// TwinCAT 3 PLC project TwinCAT_OpenFramework_Temporary
// Title: Temporary project for old code storing
// Company: Oleksandr Tiutyk FOP
// ProjectVersion: 0.0.0.1
// Description: Temporary project that contains legacy functionality and needs to be reconsidered and migrated in light of the new concepts
// ProgramVersion: 3.1.4026.16
// project tree:
//   Communication/ADS/ AdsCommunicationSettings.TcPOU, AdsCommunicator.TcPOU, ADS_COMMUNICATOR_STATE.TcDUT, ADS_REQUEST_ITEM.TcDUT
//   Communication/ CommunicationSettings.TcPOU, Communicator.TcPOU, CommunicatorSFC.TcPOU, CurrentNamespace_1.TcGVL
//   Communication/OPC_UA/ OpcUaCommunicationSettings.TcPOU, OpcUaCommunicator.TcPOU, OpcUaHelper.TcPOU, OPC_UA_ACTION_EXECUTION_STATE.TcDUT, OPC_UA_COMMUNICATOR_STATE.TcDUT
//   Communication/OPC_UA/RequestItems/ OpcUaDAReadRequestItem.TcPOU, OpcUaDARequestItem.TcPOU, OpcUaDAWriteRequestItem.TcPOU, OpcUaMethodCallRequestItem.TcPOU, OpcUaRequestItem.TcPOU, OPC_UA_OUTPUT_ARGUMENT_INFO_AND_DATA.TcDUT
//   Communication/S7/ GetStringSizeForS7Comm.TcPOU, S7CommunicationSettings.TcPOU, S7Communicator.TcPOU, S7_COMMUNICATOR_STATE.TcDUT, S7_VARIABLE.TcDUT
//   Database/Command/ DbCommandExecutor.TcPOU, DB_COMMAND_DISCONNECTING_STATE.TcDUT, DB_COMMAND_EXECUTION_PARAMETERS.TcDUT, DB_COMMAND_EXECUTION_STATE.TcDUT
//   Database/ CurrentNamespace.TcGVL
//   Database/StoredProcedure/ DbProcedureExecutor.TcPOU, DB_PROCEDURE_DISCONNECTING_STATE.TcDUT, DB_PROCEDURE_EXECUTION_STATE.TcDUT, DB_ROCEDURE_EXECUTION_PARAMETERS.TcDUT
//   Files/ CreateDirectory.TcPOU, DeleteDirectory.TcPOU, DeleteFile.TcPOU, LoadFile.TcPOU, RenameFile.TcPOU
//   Files/FileContentManager/Enums/ FILE_CONTENT_HANDLING_MODE.TcDUT, FILE_MOVE_POINTER_TYPE.TcDUT, FILE_OPEN_MODE.TcDUT
//   Files/FileContentManager/ FileContentManager.TcPOU, FileContentTask.TcPOU
//   Files/FileContentManager/Tasks/ FileCloseTask.TcPOU, FileFlushTask.TcPOU, FileGetCurrentPositionTask.TcPOU, FileMovePointerTask.TcPOU, FileOpenTask.TcPOU, FileReadBytesTask.TcPOU, FileReadStringTask.TcPOU, FileTestForEndTask.TcPOU, FileWriteBytesTask.TcPOU, FileWriteStringTask.TcPOU
//   StateMachine/Finite/ FiniteStateMachine.TcPOU, ProgramState.TcPOU, ProgramTransition.TcPOU
//   StateMachine/ ProgramConstants.TcGVL
//   StateMachine/Program/ ProgramStateMachine.TcPOU
//   StateMachine/Program/States/ HaltedProgramState.TcPOU, ReadyProgramState.TcPOU, RunningProgramState.TcPOU, SuspendedProgramState.TcPOU
//   StateMachine/Program/Transitions/ HaltedToReadyProgramTransition.TcPOU, ReadyToHaltedProgramTransition.TcPOU, ReadyToRunningProgramTransition.TcPOU, RunningToHaltedProgramTransition.TcPOU, RunningToReadyProgramTransition.TcPOU, RunningToSuspendedProgramTransition.TcPOU, SuspendedToHaltedProgramTransition.TcPOU, SuspendedToReadyProgramTransition.TcPOU, SuspendedToRunningProgramTransition.TcPOU
//   StateMachine/UnifiedProgram/States/ HaltedUnifiedProgramState.TcPOU, ReadyUnifiedProgramState.TcPOU, RunningUnifiedProgramState.TcPOU, SuspendedUnifiedProgramState.TcPOU
//   StateMachine/UnifiedProgram/StepModels/ UnifiedProgramExecutedStep.TcPOU, UnifiedProgramExecutedStepAction.TcPOU, UnifiedProgramExecutedStepHelper.TcPOU, UnifiedProgramExecutedStepTransition.TcPOU, UnifiedProgramExecutedStepTransitionCondition.TcPOU
//   StateMachine/UnifiedProgram/Steps/ UNIFIED_PROGRAM_CONFIGURATION.TcDUT, UNIFIED_PROGRAM_EXECUTED_STEP.TcDUT, UNIFIED_PROGRAM_STEP.TcDUT, UNIFIED_PROGRAM_STEP_ACTION.TcDUT, UNIFIED_PROGRAM_STEP_TRANSITION.TcDUT, UNIFIED_PROGRAM_STEP_TRANSITION_CONDITION.TcDUT
//   StateMachine/UnifiedProgram/Transitions/ HaltedToReadyUnifiedProgramTransition.TcPOU, ReadyToHaltedUnifiedProgramTransition.TcPOU, ReadyToRunningUnifiedProgramTransition.TcPOU, RunningToHaltedUnifiedProgramTransition.TcPOU, RunningToReadyUnifiedProgramTransition.TcPOU, RunningToSuspendedUnifiedProgramTransition.TcPOU, SuspendedToHaltedUnifiedProgramTransition.TcPOU, SuspendedToReadyUnifiedProgramTransition.TcPOU, SuspendedToRunningUnifiedProgramTransition.TcPOU
//   StateMachine/UnifiedProgram/ UnifiedProgramConstants.TcGVL, UnifiedProgramStateMachine.TcPOU, UnifiedProgramStepExecutor.TcPOU
//   Tasks/ SequentialTaskExecutor.TcPOU, Task.TcPOU

// ---- Communication/ADS/ADS_COMMUNICATOR_STATE.TcDUT
{attribute 'qualified_only'}
{attribute 'strict'}
{attribute 'to_string'}
TYPE ADS_COMMUNICATOR_STATE :
(
	IDLE_OR_DONE,
	READ_SYMBOL_INFO,
	DATA_PROCESSING,
	WAIT_FOR_NEXT_CYCLE
);
END_TYPE

// ---- Communication/ADS/ADS_REQUEST_ITEM.TcDUT
{attribute 'enable_dynamic_creation'}	
TYPE ADS_REQUEST_ITEM :
STRUCT
	ReadSymbolInfo : Tc2_Utilities.PLC_ReadSymInfoByName;
	ReadMode : BOOL;
	Read : Tc2_System.ADSREADEX;
	Write : Tc2_System.ADSWRITE;
	IndexGroupAndOffsetValid : BOOL;	
	ReceivedBytesCountTarget : POINTER TO UDINT;
END_STRUCT
END_TYPE

// ---- Communication/OPC_UA/OPC_UA_ACTION_EXECUTION_STATE.TcDUT
{attribute 'qualified_only'}
{attribute 'strict'}
{attribute 'to_string'}
TYPE OPC_UA_ACTION_EXECUTION_STATE :
(
	BUSY,
	DONE,
	ERROR
);
END_TYPE

// ---- Communication/OPC_UA/OPC_UA_COMMUNICATOR_STATE.TcDUT
{attribute 'qualified_only'}
{attribute 'strict'}
{attribute 'to_string'}
TYPE OPC_UA_COMMUNICATOR_STATE :
(
	IDLE,
	CONNECT,
	GET_NAMESPACE_INDEX,
	GET_NODE_HANDLE,
	PERFORM_ACTION,
	WAIT_FOR_NEXT_CYCLE,
	RELEASE_NODE_HANDLE,
	DISCONNECT
);
END_TYPE

// ---- Communication/OPC_UA/RequestItems/OPC_UA_OUTPUT_ARGUMENT_INFO_AND_DATA.TcDUT
{attribute 'pack_mode' := '1'}
TYPE OPC_UA_OUTPUT_ARGUMENT_INFO_AND_DATA :
STRUCT
	nNumberOfOutputArguments: UDINT; // determined amount of output parameters
	nReserved: ARRAY[1..4] OF BYTE; // Reserved padding
	//stOutputArgInfo: ARRAY[*] OF ST_UAMethodArgInfo; 
	//data : DINT;
END_STRUCT
END_TYPE

// ---- Communication/S7/S7_COMMUNICATOR_STATE.TcDUT
{attribute 'qualified_only'}
{attribute 'strict'}
{attribute 'to_string'}
TYPE S7_COMMUNICATOR_STATE :
(
	IDLE_OR_DONE,
	DATA_PROCESSING,
	WAIT_FOR_NEXT_CYCLE
);
END_TYPE

// ---- Communication/S7/S7_VARIABLE.TcDUT
{attribute 'enable_dynamic_creation'}	
TYPE S7_VARIABLE :
STRUCT
	Address : PVOID;
	Write : BOOL;
END_STRUCT
END_TYPE

// ---- Database/Command/DB_COMMAND_DISCONNECTING_STATE.TcDUT
{attribute 'qualified_only'}
{attribute 'strict'}
{attribute 'to_string'}
TYPE DB_COMMAND_DISCONNECTING_STATE :
(
	IDLING,
	DATA_SET_RELEASING,
	DISCONNECTING
);
END_TYPE

// ---- Database/Command/DB_COMMAND_EXECUTION_PARAMETERS.TcDUT
{attribute 'enable_dynamic_creation'}	
TYPE DB_COMMAND_EXECUTION_PARAMETERS :
STRUCT
	DbId : UDINT;
	CommandText : Tc2_System.T_MaxString;
	TargetBuffer : PVOID; 
	TargetBufferSize : UDINT;
	MaxRecordsToReadAtTime : UINT;
END_STRUCT
END_TYPE

// ---- Database/Command/DB_COMMAND_EXECUTION_STATE.TcDUT
{attribute 'qualified_only'}
{attribute 'strict'}
{attribute 'to_string'}
TYPE DB_COMMAND_EXECUTION_STATE :
(
	IDLING,
	STARTING,
	CONNECTING,
	PREPARING,
	EXECUTING,
	LOADING_RESULT_DATA_SET,
	DISCONNECTING 
);
END_TYPE

// ---- Database/StoredProcedure/DB_PROCEDURE_DISCONNECTING_STATE.TcDUT
{attribute 'qualified_only'}
{attribute 'strict'}
{attribute 'to_string'}
TYPE DB_PROCEDURE_DISCONNECTING_STATE :
(
	IDLING,
	DATA_SET_RELEASING,
	PARAMETERS_RELEASING,
	DISCONNECTING
);
END_TYPE

// ---- Database/StoredProcedure/DB_PROCEDURE_EXECUTION_STATE.TcDUT
{attribute 'qualified_only'}
{attribute 'strict'}
{attribute 'to_string'}
TYPE DB_PROCEDURE_EXECUTION_STATE :
(
	IDLING,
	STARTING,
	CONNECTING,
	PREPARING,
	EXECUTING,
	LOADING_RESULT_DATA_SET,
	DISCONNECTING
);
END_TYPE

// ---- Database/StoredProcedure/DB_ROCEDURE_EXECUTION_PARAMETERS.TcDUT
{attribute 'enable_dynamic_creation'}	
TYPE DB_ROCEDURE_EXECUTION_PARAMETERS :
STRUCT
	DbId : UDINT;
	ProcedureName : Tc2_System.T_MaxString;
	ParameterDescriptors : POINTER TO Tc3_Database.ST_SQLSPParameter;
	ParameterDescriptorsSize : UDINT;
	ParameterValues : PVOID;
	ParameterValuesSize : UDINT;	
	TargetBuffer : PVOID; 
	TargetBufferSize : UDINT;
	MaxRecordsToReadAtTime : UINT;
END_STRUCT
END_TYPE

// ---- Files/FileContentManager/Enums/FILE_CONTENT_HANDLING_MODE.TcDUT
{attribute 'qualified_only'}
{attribute 'strict'}
{attribute 'to_string'}
TYPE FILE_CONTENT_HANDLING_MODE :
(
	BINARY := Tc2_System.FOPEN_MODEBINARY, // opens the file in binary mode
	TEXT := Tc2_System.FOPEN_MODETEXT // opens the file in text mode
) DWORD;
END_TYPE

// ---- Files/FileContentManager/Enums/FILE_MOVE_POINTER_TYPE.TcDUT
{attribute 'qualified_only'}
{attribute 'strict'}
{attribute 'to_string'}
TYPE FILE_MOVE_POINTER_TYPE :
(
	FROM_FILE_BEGINNING,
	FROM_CURRENT_POSITION,
	FROM_FILE_END
);
END_TYPE

// ---- Files/FileContentManager/Enums/FILE_OPEN_MODE.TcDUT
{attribute 'qualified_only'}
{attribute 'strict'}
{attribute 'to_string'}
TYPE FILE_OPEN_MODE :
(
	READ_EXISTING := Tc2_System.FOPEN_MODEREAD, // opens a file for reading. An error is returned if the file cannot be found or does not exist
	WRITE_EMPTY := Tc2_System.FOPEN_MODEWRITE, // opens an empty file for writing. If the file already exists, it is overwritten
	APPEND := Tc2_System.FOPEN_MODEAPPEND, // opens a file for writing at the end of the file (append). If the file does not exist, a new file is created
	READ_AND_WRITE_EXISTING := Tc2_System.FOPEN_MODEREAD OR Tc2_System.FOPEN_MODEPLUS, // opens a file for reading and writing. The file must exist
	READ_AND_WRITE_EMPTY := Tc2_System.FOPEN_MODEWRITE OR Tc2_System.FOPEN_MODEPLUS, // opens an empty file FOR reading AND writing. IF the file already exists, it is overwritten.
	READ_AND_APPEND := Tc2_System.FOPEN_MODEAPPEND OR Tc2_System.FOPEN_MODEPLUS // opens a file for reading and writing at the end of the file (append). If the file does not exist, a new file is created. For this, the memory path must be known, otherwise error 1804 appears.
) DWORD;
END_TYPE

// ---- StateMachine/UnifiedProgram/Steps/UNIFIED_PROGRAM_CONFIGURATION.TcDUT
TYPE UNIFIED_PROGRAM_CONFIGURATION :
STRUCT
	Name : STRING(255) := 'New program';
	Version : DATE_AND_TIME;
	Steps : ARRAY [0..UnifiedProgramConstants.MaxStepCount - 1] OF UNIFIED_PROGRAM_STEP;
END_STRUCT
END_TYPE

// ---- StateMachine/UnifiedProgram/Steps/UNIFIED_PROGRAM_EXECUTED_STEP.TcDUT
TYPE UNIFIED_PROGRAM_EXECUTED_STEP :
STRUCT
	StepIndex : INT := -1;
	
	Step : REFERENCE TO UNIFIED_PROGRAM_STEP;
END_STRUCT
END_TYPE

// ---- StateMachine/UnifiedProgram/Steps/UNIFIED_PROGRAM_STEP.TcDUT
TYPE UNIFIED_PROGRAM_STEP :
STRUCT
	Suspend : BOOL;
	Complete : BOOL;
	Actions : ARRAY [0..UnifiedProgramConstants.MaxStepActionsCount - 1] OF UNIFIED_PROGRAM_STEP_ACTION;
	Transitions : ARRAY [0..UnifiedProgramConstants.MaxStepTransitionsCount - 1] OF UNIFIED_PROGRAM_STEP_TRANSITION;
END_STRUCT
END_TYPE

// ---- StateMachine/UnifiedProgram/Steps/UNIFIED_PROGRAM_STEP_ACTION.TcDUT
TYPE UNIFIED_PROGRAM_STEP_ACTION :
STRUCT
	Name : STRING;
	Args : ARRAY [0..UnifiedProgramConstants.MaxActionArgumentsCount - 1] OF STRING(255);
END_STRUCT
END_TYPE

// ---- StateMachine/UnifiedProgram/Steps/UNIFIED_PROGRAM_STEP_TRANSITION.TcDUT
TYPE UNIFIED_PROGRAM_STEP_TRANSITION :
STRUCT
	Condition : UNIFIED_PROGRAM_STEP_TRANSITION_CONDITION;
	Target : BYTE;
END_STRUCT
END_TYPE

// ---- StateMachine/UnifiedProgram/Steps/UNIFIED_PROGRAM_STEP_TRANSITION_CONDITION.TcDUT
TYPE UNIFIED_PROGRAM_STEP_TRANSITION_CONDITION :
STRUCT
	Name : STRING;
	Args : ARRAY [0..UnifiedProgramConstants.MaxActionArgumentsCount - 1] OF STRING(255);
END_STRUCT
END_TYPE

// ---- Communication/CurrentNamespace_1.TcGVL
{attribute 'qualified_only'}
VAR_GLOBAL
	{attribute 'OPC.UA.DA' := '1'}
	{attribute 'OPC.UA.DA.Access' := '1'}
	{attribute 'init_namespace'} 
	Name : STRING(255);	
END_VAR

// ---- Database/CurrentNamespace.TcGVL
{attribute 'qualified_only'}
VAR_GLOBAL
	{attribute 'OPC.UA.DA' := '1'}
	{attribute 'OPC.UA.DA.Access' := '1'}
	{attribute 'init_namespace'} 
	Name : STRING(255);	
END_VAR

// ---- StateMachine/ProgramConstants.TcGVL
{attribute 'qualified_only'}
VAR_GLOBAL CONSTANT
	MaxStateCount : INT := 5;
	MaxTransitionCount : INT := 20;
END_VAR

// ---- StateMachine/UnifiedProgram/UnifiedProgramConstants.TcGVL
{attribute 'qualified_only'}
VAR_GLOBAL CONSTANT
	MaxStepCount : INT := 5;	
	MaxStepActionsCount : INT := 5;
	MaxStepTransitionsCount : INT := 2;
	MaxActionArgumentsCount : INT := 5;
	MaxConditionArgumentsCount : INT := 5;
END_VAR

// ---- Communication/ADS/AdsCommunicationSettings.TcPOU
{attribute 'no_explicit_call' := 'do not call this function block directly'} 
FUNCTION_BLOCK AdsCommunicationSettings EXTENDS CommunicationSettings
VAR_INPUT
	AmsNetId : Tc2_System.T_AmsNetID;
	AmsPort : Tc2_System.T_AmsPort := 801;
END_VAR
VAR
	_ClassName : STRING := __POUNAME();
END_VAR

PROPERTY CommunicationTypeName : STRING
GET
CommunicationTypeName := 'ADS';
END_GET
END_PROPERTY

END_FUNCTION_BLOCK

// ---- Communication/CommunicationSettings.TcPOU
FUNCTION_BLOCK ABSTRACT CommunicationSettings
VAR_INPUT
	DefaultOperationTimeout : TIME := Tc2_System.DEFAULT_ADS_TIMEOUT;
END_VAR

PROPERTY ABSTRACT CommunicationTypeName : STRING
GET
END_GET
END_PROPERTY

END_FUNCTION_BLOCK

// ---- Communication/ADS/AdsCommunicator.TcPOU
{attribute 'no_explicit_call' := 'do not call this function block directly'} 
FUNCTION_BLOCK AdsCommunicator EXTENDS Communicator
VAR
	{attribute 'OPC.UA.DA' := '0'}	
	_ClassName : STRING := __POUNAME();

	{attribute 'OPC.UA.DA' := '0'}	
	_State : ADS_COMMUNICATOR_STATE;
	{attribute 'OPC.UA.DA' := '0'}	
	_DataProcessed : BOOL;

	{attribute 'OPC.UA.DA' := '0'}
	_Items : List(POINTER_TYPE.STRUCT_POINTER); // of ADS_REQUEST_ITEM 

	{attribute 'OPC.UA.DA' := '0'}	
	_OperationTimer : Timer;	
END_VAR

METHOD AddReadByIndexGroupAndOffset : DINT
VAR_INPUT
	indexGroup : UDINT;
	indexOffset : UDINT;
	targetVariable : __SYSTEM.AnyType;
	receivedBytesCountTarget : POINTER TO UDINT;
	operationTimeout : TIME := T#0S;
END_VAR
VAR_OUTPUT
	exception : Exception;
END_VAR
VAR
	request : POINTER TO ADS_REQUEST_ITEM;
END_VAR
AddReadByIndexGroupAndOffset := -1;

IF Busy THEN
	ExceptionHelper.Throw(0, "AdsRequest is already executing", __POUNAME(), ClassName, CurrentNamespace.Name, __POSITION());
	RETURN;
END_IF

request := __NEW(ADS_REQUEST_ITEM);

request^.ReadMode := TRUE;
request^.ReadSymbolInfo.SYMNAME := '';
request^.Read.IDXGRP := indexGroup;
request^.Read.IDXOFFS := indexOffset;
request^.Read.DESTADDR := targetVariable.pValue;
request^.Read.LEN := TO_UDINT(targetVariable.diSize);
request^.Read.TMOUT := GetOperationTimeout(operationTimeout);
request^.IndexGroupAndOffsetValid := TRUE;
request^.ReceivedBytesCountTarget := receivedBytesCountTarget;

AddReadByIndexGroupAndOffset := _Items.Append(request);
END_METHOD

METHOD AddReadBySymbolName : DINT
VAR_INPUT
	symbolName : Tc2_System.T_MaxString;
	targetVariable : __SYSTEM.AnyType;
	receivedBytesCountTarget : POINTER TO UDINT;
	operationTimeout : TIME := T#0S;
END_VAR
VAR_OUTPUT
	exception : Exception;
END_VAR
VAR
	request : POINTER TO ADS_REQUEST_ITEM;
END_VAR
AddReadBySymbolName := -1;

IF Busy THEN
	ExceptionHelper.Throw(0, "AdsRequest is already executing", __POUNAME(), ClassName, CurrentNamespace.Name, __POSITION());
	RETURN;
END_IF

IF SymbolName = '' THEN
	ExceptionHelper.Throw(0, "Parameter 'symbolName' is not specified", __POUNAME(), ClassName, CurrentNamespace.Name, __POSITION());
	RETURN;
END_IF

request := __NEW(ADS_REQUEST_ITEM);

request^.ReadMode := TRUE;
request^.ReadSymbolInfo.SYMNAME := symbolName;
request^.Read.IDXGRP := 0;
request^.Read.IDXOFFS := 0;
request^.Read.DESTADDR := targetVariable.pValue;
request^.Read.LEN := TO_UDINT(targetVariable.diSize);
request^.Read.TMOUT := GetOperationTimeout(operationTimeout);
request^.IndexGroupAndOffsetValid := FALSE;
request^.ReceivedBytesCountTarget := receivedBytesCountTarget;

AddReadBySymbolName := _Items.Append(request);
END_METHOD

METHOD AddWriteByIndexGroupAndOffset : DINT
VAR_INPUT
	indexGroup : UDINT;
	indexOffset : UDINT;
	sourceVariable : __SYSTEM.AnyType;
	operationTimeout : TIME := T#0S;
END_VAR
VAR_OUTPUT
	exception : Exception;
END_VAR
VAR
	request : POINTER TO ADS_REQUEST_ITEM;
END_VAR
AddWriteByIndexGroupAndOffset := -1;

IF Busy THEN
	ExceptionHelper.Throw(0, "AdsRequest is already executing", __POUNAME(), ClassName, CurrentNamespace.Name, __POSITION());
	RETURN;
END_IF

request := __NEW(ADS_REQUEST_ITEM);

request^.ReadMode := FALSE;
request^.ReadSymbolInfo.SYMNAME := '';
request^.Write.IDXGRP := indexGroup;
request^.Write.IDXOFFS := indexOffset;
request^.Write.SRCADDR := sourceVariable.pValue;
request^.Write.LEN := TO_UDINT(sourceVariable.diSize);
request^.Write.TMOUT := GetOperationTimeout(operationTimeout);
request^.IndexGroupAndOffsetValid := TRUE;

AddWriteByIndexGroupAndOffset := _Items.Append(request);
END_METHOD

METHOD AddWriteBySymbolName : DINT
VAR_INPUT
	symbolName : Tc2_System.T_MaxString;
	sourceVariable : __SYSTEM.AnyType;
	operationTimeout : TIME := T#0S;
END_VAR
VAR_OUTPUT
	exception : Exception;
END_VAR
VAR
	request : POINTER TO ADS_REQUEST_ITEM;
END_VAR
AddWriteBySymbolName := -1;

IF Busy THEN
	ExceptionHelper.Throw(0, "AdsRequest is already executing", __POUNAME(), ClassName, CurrentNamespace.Name, __POSITION());
	RETURN;
END_IF

IF SymbolName = '' THEN
	ExceptionHelper.Throw(0, "Parameter 'symbolName' is not specified", __POUNAME(), ClassName, CurrentNamespace.Name, __POSITION());
	RETURN;
END_IF

request := __NEW(ADS_REQUEST_ITEM);

request^.ReadMode := FALSE;
request^.ReadSymbolInfo.SYMNAME := symbolName;
request^.Write.IDXGRP := 0;
request^.Write.IDXOFFS := 0;
request^.Write.SRCADDR := sourceVariable.pValue;
request^.Write.LEN := TO_UDINT(sourceVariable.diSize);
request^.Write.TMOUT := GetOperationTimeout(operationTimeout);
request^.IndexGroupAndOffsetValid := FALSE;

AddWriteBySymbolName := _Items.Append(request);
END_METHOD

{attribute 'monitoring' := 'call'}
{attribute 'OPC.UA.DA' := '1'}
{attribute 'OPC.UA.DA.Property' := '1'}
PROPERTY Busy : BOOL
GET
Busy := _LastException.Empty AND_THEN _State <> ADS_COMMUNICATOR_STATE.IDLE_OR_DONE;
END_GET
END_PROPERTY

{attribute 'monitoring' := 'call'}
PROPERTY ClassName : STRING
GET
ClassName := _ClassName;
END_GET
END_PROPERTY

PROPERTY CommunicationTypeName : STRING
GET
CommunicationTypeName := 'ADS';
END_GET
END_PROPERTY

{attribute 'monitoring' := 'call'}
{attribute 'OPC.UA.DA' := '1'}
{attribute 'OPC.UA.DA.Property' := '1'}
PROPERTY DataProcessed : BOOL
GET
DataProcessed := _DataProcessed;
END_GET
END_PROPERTY

{attribute 'monitoring' := 'call'}
{attribute 'OPC.UA.DA' := '1'}
{attribute 'OPC.UA.DA.Property' := '1'}
PROPERTY Error : BOOL
GET
Error := NOT _LastException.Empty;
END_GET
END_PROPERTY

METHOD Execute 
VAR
	i : DINT;
	readyItemsCount : DINT;
	item : POINTER TO ADS_REQUEST_ITEM;
END_VAR
_DataProcessed := FALSE;
_OperationTimer.Execute();

StateMachine:

readyItemsCount := 0;

CASE _State OF
	ADS_COMMUNICATOR_STATE.READ_SYMBOL_INFO:
		FOR i := 0 TO _Items.Count - 1 DO
			item := _Items.Get(i); 
			
			IF NOT item^.IndexGroupAndOffsetValid THEN
				item^.ReadSymbolInfo(START := TRUE);
				
				IF item^.ReadSymbolInfo.ERR THEN
					_LastExceptionHelper.Throw(item^.ReadSymbolInfo.ERRID, WStringHelper.Concat2("Execution of PLC_ReadSymInfoByName failed with error id = ", TO_WSTRING(item^.ReadSymbolInfo.ERRID)), __POUNAME(), ClassName, CurrentNamespace.Name, __POSITION());	
					_State := ADS_COMMUNICATOR_STATE.IDLE_OR_DONE;
					RETURN;
				ELSIF NOT item^.ReadSymbolInfo.BUSY THEN
					IF item^.ReadMode THEN
						item^.Read.IDXGRP := item^.ReadSymbolInfo.SYMINFO.idxGroup;
						item^.Read.IDXOFFS := item^.ReadSymbolInfo.SYMINFO.idxOffset;
					ELSE
						item^.Write.IDXGRP := item^.ReadSymbolInfo.SYMINFO.idxGroup;
						item^.Write.IDXOFFS := item^.ReadSymbolInfo.SYMINFO.idxOffset;
					END_IF		

					item^.IndexGroupAndOffsetValid := TRUE;	
					readyItemsCount := readyItemsCount + 1;
				END_IF
			ELSE
				readyItemsCount := readyItemsCount + 1;
			END_IF
		END_FOR
		
		IF readyItemsCount = _Items.Count THEN	
			_State := ADS_COMMUNICATOR_STATE.DATA_PROCESSING;				
			_OperationTimer.Start();
			JMP StateMachine;
		END_IF		
		
	ADS_COMMUNICATOR_STATE.DATA_PROCESSING:
		FOR i := 0 TO _Items.Count - 1 DO
			item := _Items.Get(i); 
			
			IF item^.ReadMode THEN
				item^.Read(READ := TRUE);
				
				IF item^.Read.ERR THEN
					_LastExceptionHelper.Throw(item^.Read.ERRID, WStringHelper.Concat2("Execution of ADSREADEX failed with error id = ", TO_WSTRING(item^.Read.ERRID)), __POUNAME(), ClassName, CurrentNamespace.Name, __POSITION());
					_State := ADS_COMMUNICATOR_STATE.IDLE_OR_DONE;
					RETURN;
				ELSIF NOT item^.Read.BUSY THEN
					IF item^.ReceivedBytesCountTarget <> 0 THEN
						item^.ReceivedBytesCountTarget^ := item^.Read.COUNT_R;
					END_IF
					
					readyItemsCount := readyItemsCount + 1;
				END_IF
			ELSE
				item^.Write(WRITE := TRUE);
				
				IF item^.Write.ERR THEN
					_LastExceptionHelper.Throw(item^.Write.ERRID, WStringHelper.Concat2("Execution of ADSWRITE failed with error id = ", TO_WSTRING(item^.Write.ERRID)), __POUNAME(), ClassName, CurrentNamespace.Name, __POSITION());
					_State := ADS_COMMUNICATOR_STATE.IDLE_OR_DONE;
					RETURN;
				ELSIF NOT item^.Write.BUSY THEN
					readyItemsCount := readyItemsCount + 1;
				END_IF
			END_IF
		END_FOR
		
		IF readyItemsCount = _Items.Count THEN
			_DataProcessed := TRUE;	
			CycleCount := CycleCount + 1;
			
			IF CyclicMode THEN
				_State := ADS_COMMUNICATOR_STATE.WAIT_FOR_NEXT_CYCLE;	
				JMP StateMachine;			
			ELSE	
				_State := ADS_COMMUNICATOR_STATE.IDLE_OR_DONE;		
			END_IF
		END_IF	
		
	ADS_COMMUNICATOR_STATE.WAIT_FOR_NEXT_CYCLE:
		IF _OperationTimer.ElapsedTime >= CycleInterval THEN
			FOR i := 0 TO _Items.Count - 1 DO
				item := _Items.Get(i); 
				
				IF item^.ReadMode THEN
					item^.Read(READ := FALSE);
				ELSE
					item^.Write(WRITE := FALSE);
				END_IF
			END_FOR	
			
			_State := ADS_COMMUNICATOR_STATE.DATA_PROCESSING;
			_OperationTimer.Start();			
			JMP StateMachine;	
		END_IF
END_CASE
END_METHOD

METHOD FB_exit : BOOL
VAR_INPUT
	bInCopyCode : BOOL; // if TRUE, the exit method is called for exiting an instance that is copied afterwards (online change).
END_VAR
_Items.Clear(TRUE);
END_METHOD

METHOD PROTECTED InternalClear : BOOL
VAR_OUTPUT
	exception : Exception;
END_VAR
_Items.Clear(TRUE);

_State := ADS_COMMUNICATOR_STATE.IDLE_OR_DONE;

InternalClear := TRUE;
END_METHOD

METHOD PROTECTED InternalConfigure : BOOL
VAR_INPUT
	settings : REFERENCE TO CommunicationSettings;
END_VAR
VAR_OUTPUT
	exception : Exception;
END_VAR
VAR
	adsSettings : POINTER TO AdsCommunicationSettings;
	i : DINT;
	item : POINTER TO ADS_REQUEST_ITEM;
END_VAR
adsSettings := ADR(settings);

_OperationTimer.Interval := T#1H;

IF adsSettings^.AmsPort = 0 THEN
	ExceptionHelper.Throw(0, "settings.AmsPort is not specified", __POUNAME(), ClassName, CurrentNamespace.Name, __POSITION());
	RETURN;
END_IF

FOR i := 0 TO _Items.Count - 1 DO
	item := _Items.Get(i);
	
	item^.ReadSymbolInfo(NETID := adsSettings^.AmsNetId, PORT := adsSettings^.AmsPort);		
	item^.Read(NETID := adsSettings^.AmsNetId, PORT := adsSettings^.AmsPort);
	item^.Write(NETID := adsSettings^.AmsNetId, PORT := adsSettings^.AmsPort);
END_FOR

InternalConfigure := TRUE;
END_METHOD

METHOD PROTECTED InternalStart : BOOL
VAR_OUTPUT
	exception : Exception;
END_VAR
VAR
	i : DINT;
	item : POINTER TO ADS_REQUEST_ITEM;
END_VAR
_State := ADS_COMMUNICATOR_STATE.READ_SYMBOL_INFO;

FOR i := 0 TO _Items.Count - 1 DO
	item := _Items.Get(i);
	
	item^.ReadSymbolInfo(START := FALSE);	
	
	IF item^.ReadMode THEN
		item^.Read(READ := FALSE);
	ELSE
		item^.Write(WRITE := FALSE);
	END_IF
END_FOR

InternalStart := TRUE;
END_METHOD

METHOD PROTECTED InternalStop
_State := ADS_COMMUNICATOR_STATE.IDLE_OR_DONE;
_OperationTimer.Stop();
END_METHOD

PROPERTY VariablesCount : DINT
GET
VariablesCount := _Items.Count;
END_GET
END_PROPERTY

END_FUNCTION_BLOCK

// ---- Communication/Communicator.TcPOU
FUNCTION_BLOCK ABSTRACT Communicator EXTENDS TC.ToolkitObject
VAR_INPUT
	CycleInterval : TIME; 
	CyclicMode : BOOL; 
END_VAR
VAR_OUTPUT
	{attribute 'OPC.UA.DA.Access' := '1'}	
	Configured : BOOL;
	{attribute 'OPC.UA.DA.Access' := '1'}	
	CycleCount : ULINT;
	{attribute 'OPC.UA.DA.Access' := '1'}	
	DefaultOperationTimeout : TIME; 
END_VAR
VAR
	{attribute 'OPC.UA.DA' := '0'}	
	_InitialCyclicMode : BOOL; 
	{attribute 'OPC.UA.DA' := '0'}	
	_LastException : Exception;
END_VAR

{attribute 'monitoring' := 'call'}
{attribute 'OPC.UA.DA' := '1'}
{attribute 'OPC.UA.DA.Property' := '1'}
PROPERTY ABSTRACT Busy : BOOL
GET
END_GET
END_PROPERTY

METHOD Clear : BOOL
VAR_OUTPUT
	exception : Exception;
END_VAR
IF Busy THEN
	ExceptionHelper.Throw(0, "Communicator is busy", __POUNAME(), ClassName, CurrentNamespace.Name, __POSITION());
	RETURN;
END_IF

AdsLogger.LogMessage(LOGGING_LEVEL.INFORMATION, "---Communicator.Clear");

CycleCount := 0;
_LastException.Clear();

Clear := InternalClear(exception => exception);
END_METHOD

PROPERTY ABSTRACT CommunicationTypeName : STRING
GET
END_GET
END_PROPERTY

METHOD FINAL Configure : BOOL
VAR_INPUT
	settings : REFERENCE TO CommunicationSettings;
END_VAR
VAR_OUTPUT
	exception : Exception;
END_VAR
IF Busy THEN
	ExceptionHelper.Throw(0, "Communicator is busy", __POUNAME(), ClassName, CurrentNamespace.Name, __POSITION());
	RETURN;
END_IF

IF NOT __ISVALIDREF(settings) THEN
	ExceptionHelper.Throw(0, "Parameter 'settings' has not been specified", __POUNAME(), ClassName, CurrentNamespace.Name, __POSITION());
	RETURN;
END_IF

IF CommunicationTypeName <> settings.CommunicationTypeName THEN
	ExceptionHelper.Throw(0, WStringHelper.Concat4("Communicator and communication settings are incompatible because has different CommunicationTypeName: ", TO_WSTRING(CommunicationTypeName), " and ", TO_WSTRING(settings.CommunicationTypeName)), __POUNAME(), ClassName, CurrentNamespace.Name, __POSITION());
	RETURN;
END_IF

IF settings.DefaultOperationTimeout > T#0S THEN
	DefaultOperationTimeout := settings.DefaultOperationTimeout;
ELSE	
	DefaultOperationTimeout := Tc2_System.DEFAULT_ADS_TIMEOUT;
END_IF

AdsLogger.LogMessage(LOGGING_LEVEL.INFORMATION, "---Communicator.Configure");

Configured := Configure := InternalConfigure(settings, exception => exception);
END_METHOD

{attribute 'monitoring' := 'call'}
{attribute 'OPC.UA.DA' := '1'}
{attribute 'OPC.UA.DA.Property' := '1'}
PROPERTY DataProcessed : BOOL
GET
END_GET
END_PROPERTY

{attribute 'monitoring' := 'call'}
{attribute 'OPC.UA.DA' := '1'}
{attribute 'OPC.UA.DA.Property' := '1'}
PROPERTY Error : BOOL
GET
END_GET
END_PROPERTY

METHOD ABSTRACT Execute
END_METHOD

METHOD PROTECTED GetOperationTimeout : TIME
VAR_INPUT
	operationTimeout : TIME;
END_VAR
IF operationTimeout = T#0S THEN
	getOperationTimeout := DefaultOperationTimeout;
ELSE
	getOperationTimeout := operationTimeout;
END_IF
END_METHOD

METHOD PROTECTED ABSTRACT InternalClear : BOOL
VAR_OUTPUT
	exception : Exception;
END_VAR
END_METHOD

METHOD PROTECTED ABSTRACT InternalConfigure : BOOL
VAR_INPUT
	settings : REFERENCE TO CommunicationSettings;
END_VAR
VAR_OUTPUT
	exception : Exception;
END_VAR
END_METHOD

METHOD PROTECTED ABSTRACT InternalStart : BOOL
VAR_OUTPUT
	exception : Exception;
END_VAR
END_METHOD

METHOD PROTECTED ABSTRACT InternalStop
END_METHOD

{attribute 'monitoring' := 'call'}
{attribute 'OPC.UA.DA.Property' := '1'}
{attribute 'OPC.UA.DA.Access' := '1'}
PROPERTY FINAL LastException : REFERENCE TO Exception
GET
LastException REF= _LastException;
END_GET
END_PROPERTY

METHOD FINAL Start : BOOL
VAR_OUTPUT
	exception : Exception;
END_VAR
IF Busy THEN
	ExceptionHelper.Throw(0, "Communicator is busy", __POUNAME(), ClassName, CurrentNamespace.Name, __POSITION());
	RETURN;
END_IF

AdsLogger.LogMessage(LOGGING_LEVEL.INFORMATION, "---Communicator.Start");

CycleCount := 0;
_LastException.Clear();

Start := InternalStart(exception => exception);
END_METHOD

METHOD FINAL Stop
IF Busy THEN
	AdsLogger.LogMessage(LOGGING_LEVEL.INFORMATION, "---Communicator.Stop");
		
	InternalStop();
END_IF
END_METHOD

PROPERTY ABSTRACT VariablesCount : DINT
GET
END_GET
END_PROPERTY

END_FUNCTION_BLOCK

// ---- Communication/CommunicatorSFC.TcPOU
FUNCTION_BLOCK ABSTRACT CommunicatorSFC EXTENDS TC.ToolkitObject

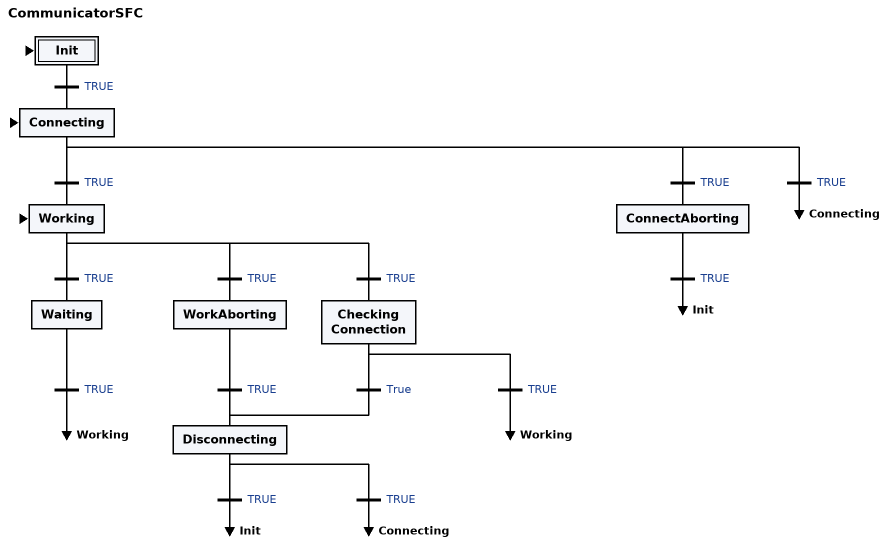
INITIAL_STEP Init:
END_STEP
TRANSITION FROM Init TO Connecting
    := TRUE;
END_TRANSITION
STEP Connecting:
END_STEP
TRANSITION FROM Connecting TO Working
    := TRUE;
END_TRANSITION
STEP Working:
END_STEP
TRANSITION FROM Connecting TO ConnectAborting
    := TRUE;
END_TRANSITION
STEP ConnectAborting:
END_STEP
TRANSITION FROM ConnectAborting TO Init
    := TRUE;
END_TRANSITION
TRANSITION FROM Connecting TO Connecting
    := TRUE;
END_TRANSITION
TRANSITION FROM Working TO Waiting
    := TRUE;
END_TRANSITION
STEP Waiting:
END_STEP
TRANSITION FROM Waiting TO Working
    := TRUE;
END_TRANSITION
TRANSITION FROM Working TO WorkAborting
    := TRUE;
END_TRANSITION
STEP WorkAborting:
END_STEP
TRANSITION FROM WorkAborting TO Disconnecting
    := TRUE;
END_TRANSITION
TRANSITION FROM Working TO CheckingConnection
    := TRUE;
END_TRANSITION
STEP CheckingConnection:
END_STEP
TRANSITION FROM CheckingConnection TO Disconnecting
    := True;
END_TRANSITION
TRANSITION FROM CheckingConnection TO Working
    := TRUE;
END_TRANSITION
STEP Disconnecting:
END_STEP
TRANSITION FROM Disconnecting TO Init
    := TRUE;
END_TRANSITION
TRANSITION FROM Disconnecting TO Connecting
    := TRUE;
END_TRANSITION

END_FUNCTION_BLOCK

// ---- Communication/OPC_UA/OpcUaCommunicationSettings.TcPOU
{attribute 'no_explicit_call' := 'do not call this function block directly'} 
FUNCTION_BLOCK OpcUaCommunicationSettings EXTENDS CommunicationSettings
VAR_INPUT
	ServerUrl : Tc2_System.T_MaxString;
	SessionConnectInfo : Tc3_PLCopen_OpcUa.ST_UASessionConnectInfo;
	ConnectionTimeout : TIME := Tc2_System.DEFAULT_ADS_TIMEOUT;
END_VAR
VAR
	_ClassName : STRING := __POUNAME();
END_VAR

PROPERTY CommunicationTypeName : STRING
GET
CommunicationTypeName := 'OPC-UA';
END_GET
END_PROPERTY

END_FUNCTION_BLOCK

// ---- Communication/OPC_UA/OpcUaCommunicator.TcPOU
{attribute 'no_explicit_call' := 'do not call this function block directly'} 
FUNCTION_BLOCK OpcUaCommunicator EXTENDS Communicator
VAR
	{attribute 'OPC.UA.DA' := '0'}	
	_ClassName : STRING := __POUNAME();

	{attribute 'OPC.UA.DA' := '0'}	
	_State : OPC_UA_COMMUNICATOR_STATE;	
	{attribute 'OPC.UA.DA' := '0'}	
	_DataProcessed : BOOL;

	{attribute 'OPC.UA.DA' := '0'}	
	_Connect : Tc3_PLCopen_OpcUa.UA_Connect;

	{attribute 'OPC.UA.DA' := '0'}
	_NamespaceUris : Dictionary(POINTER_TYPE.STRING_POINTER, POINTER_TYPE.STRUCT_POINTER, 0); // of STRING(MAX) and UA_GetNamespaceIndex

	{attribute 'OPC.UA.DA' := '0'}	
	_RequestItems : List(POINTER_TYPE.OBJECT_POINTER); // of POINTER TO OpcUaRequestItem
	
	{attribute 'OPC.UA.DA' := '0'}	
	_Disconnect : Tc3_PLCopen_OpcUa.UA_Disconnect;

	{attribute 'OPC.UA.DA' := '0'}
	_TimeoutTimer : Timer;	
	{attribute 'OPC.UA.DA' := '0'}	
	_OperationTimer : Timer;	
END_VAR

METHOD AddMethodCallByNamespaceIndex : DINT
VAR_INPUT
	objectNamespaceIndex : UINT; 
	objectIdentifierType : Tc3_PLCopen_OpcUa.E_UAIdentifierType;
	objectIdentifier : STRING(Tc2_System.MAX_STRING_LENGTH);	
	methodNamespaceIndex : UINT; 
	methodIdentifierType : Tc3_PLCopen_OpcUa.E_UAIdentifierType;
	methodIdentifier : STRING(Tc2_System.MAX_STRING_LENGTH);
	inputArgumentInfosAddress : POINTER TO ST_UAMethodArgInfo;
	inputArgumentInfosSize : UDINT;
	inputConstantArgumentsAddress : PVOID;
	inputConstantArgumentsSize : UDINT;
	inputDynamicArgumentsAddress : PVOID;
	inputDynamicArgumentsSize : UDINT;
	outputArgumentInfosAddress : POINTER TO ST_UAMethodArgInfo;
	outputArgumentInfosSize : UDINT;
	outputArgumentsInfoAndDataAddress : POINTER TO OPC_UA_OUTPUT_ARGUMENT_INFO_AND_DATA;
	outputArgumentsInfoAndDataSize : UDINT;
	numberOfReceivedBytesCount : POINTER TO UDINT;
	operationTimeout : TIME := T#0S;
END_VAR
VAR_OUTPUT
	exception : Exception;
END_VAR
VAR
	requestItem : POINTER TO OpcUaMethodCallRequestItem;
END_VAR
AddMethodCallByNamespaceIndex := -1;

IF Busy THEN
	ExceptionHelper.Throw(0, "OpcUaRequest is executing", __POUNAME(), ClassName, CurrentNamespace.Name, __POSITION());
	RETURN;
END_IF

_TimeoutTimer.Interval := _TimeoutTimer.Interval + operationTimeout;

requestItem := __NEW(OpcUaMethodCallRequestItem);

requestItem^.Initialize(
	objectNamespaceUri := '',
	objectNamespaceIndex := objectNamespaceIndex,
	objectIdentifierType := objectIdentifierType,
	objectIdentifier := objectIdentifier,	
	methodNamespaceUri := '',
	methodNamespaceIndex := methodNamespaceIndex,
	methodIdentifierType := methodIdentifierType,
	methodIdentifier := methodIdentifier,
	inputArgumentInfosAddress := inputArgumentInfosAddress,
	inputArgumentInfosSize := inputArgumentInfosSize,
	inputConstantArgumentsAddress := inputConstantArgumentsAddress,
	inputConstantArgumentsSize := inputConstantArgumentsSize,
	inputDynamicArgumentsAddress := inputDynamicArgumentsAddress,
	inputDynamicArgumentsSize := inputDynamicArgumentsSize,
	outputArgumentInfosAddress := outputArgumentInfosAddress,
	outputArgumentInfosSize := outputArgumentInfosSize,
	outputArgumentsInfoAndDataAddress := outputArgumentsInfoAndDataAddress,
	outputArgumentsInfoAndDataSize := outputArgumentsInfoAndDataSize,
	numberOfReceivedBytesCount := numberOfReceivedBytesCount,
	operationTimeout := operationTimeout
);

AddMethodCallByNamespaceIndex := _RequestItems.Append(requestItem);
END_METHOD

METHOD AddMethodCallByNamespaceUri : DINT
VAR_INPUT
	objectNamespaceUri : STRING(Tc2_System.MAX_STRING_LENGTH); 
	objectIdentifierType : Tc3_PLCopen_OpcUa.E_UAIdentifierType;
	objectIdentifier : STRING(Tc2_System.MAX_STRING_LENGTH);	
	methodNamespaceUri : STRING(Tc2_System.MAX_STRING_LENGTH); 
	methodIdentifierType : Tc3_PLCopen_OpcUa.E_UAIdentifierType;
	methodIdentifier : STRING(Tc2_System.MAX_STRING_LENGTH);
	inputArgumentInfosAddress : POINTER TO ST_UAMethodArgInfo;
	inputArgumentInfosSize : UDINT;
	inputConstantArgumentsAddress : PVOID;
	inputConstantArgumentsSize : UDINT;
	inputDynamicArgumentsAddress : PVOID;
	inputDynamicArgumentsSize : UDINT;
	outputArgumentInfosAddress : POINTER TO ST_UAMethodArgInfo;
	outputArgumentInfosSize : UDINT;
	outputArgumentsInfoAndDataAddress : POINTER TO OPC_UA_OUTPUT_ARGUMENT_INFO_AND_DATA;
	outputArgumentsInfoAndDataSize : UDINT;
	numberOfReceivedBytesCount : POINTER TO UDINT;
	operationTimeout : TIME := T#0S;
END_VAR
VAR_OUTPUT
	exception : Exception;
END_VAR
VAR
	namespaceUriPointer : POINTER TO STRING(MAX_STRING_LENGTH);
	getNamespaceIndex : POINTER TO Tc3_PLCopen_OpcUa.UA_GetNamespaceIndex;
	requestItem : POINTER TO OpcUaMethodCallRequestItem;
END_VAR
AddMethodCallByNamespaceUri := -1;

IF Busy THEN
	ExceptionHelper.Throw(0, "OpcUaRequest is executing", __POUNAME(), ClassName, CurrentNamespace.Name, __POSITION());
	RETURN;
END_IF

IF objectNamespaceUri = '' THEN
	ExceptionHelper.Throw(0, "Parameter 'objectNamespaceUri' is empty", __POUNAME(), ClassName, CurrentNamespace.Name, __POSITION());
	RETURN;	
END_IF

IF methodNamespaceUri = '' THEN
	ExceptionHelper.Throw(0, "Parameter 'methodNamespaceUri' is empty", __POUNAME(), ClassName, CurrentNamespace.Name, __POSITION());
	RETURN;	
END_IF

_TimeoutTimer.Interval := _TimeoutTimer.Interval + operationTimeout;

// try get existing object namespace index request
getNamespaceIndex := _NamespaceUris.GetValueByKey(ADR(objectNamespaceUri));

IF getNamespaceIndex <> 0 THEN
	IF operationTimeout > getNamespaceIndex^.Timeout THEN
		getNamespaceIndex^.Timeout := operationTimeout;	
	END_IF
// if not exists then create new request
ELSE
	namespaceUriPointer := __NEW(STRING(MAX_STRING_LENGTH));
	namespaceUriPointer^ := objectNamespaceUri;
	
	getNamespaceIndex := __NEW(Tc3_PLCopen_OpcUa.UA_GetNamespaceIndex);
	getNamespaceIndex^.NamespaceUri := objectNamespaceUri;
	getNamespaceIndex^.Timeout := operationTimeout;	
	
	_NamespaceUris.Set(namespaceUriPointer, getNamespaceIndex, TRUE, TRUE);
END_IF

// try get existing method namespace index request
getNamespaceIndex := _NamespaceUris.GetValueByKey(ADR(methodNamespaceUri));

IF getNamespaceIndex <> 0 THEN
	IF operationTimeout > getNamespaceIndex^.Timeout THEN
		getNamespaceIndex^.Timeout := operationTimeout;	
	END_IF
// if not exists then create new request
ELSE
	namespaceUriPointer := __NEW(STRING(MAX_STRING_LENGTH));
	namespaceUriPointer^ := methodNamespaceUri;
	
	getNamespaceIndex := __NEW(Tc3_PLCopen_OpcUa.UA_GetNamespaceIndex);
	getNamespaceIndex^.NamespaceUri := methodNamespaceUri;
	getNamespaceIndex^.Timeout := operationTimeout;	
	
	_NamespaceUris.Set(namespaceUriPointer, getNamespaceIndex, TRUE, TRUE);
END_IF

requestItem := __NEW(OpcUaMethodCallRequestItem);

requestItem^.Initialize(
	objectNamespaceUri := objectNamespaceUri,
	objectNamespaceIndex := 0,
	objectIdentifierType := objectIdentifierType,
	objectIdentifier := objectIdentifier,	
	methodNamespaceUri := methodNamespaceUri,
	methodNamespaceIndex := 0,
	methodIdentifierType := methodIdentifierType,
	methodIdentifier := methodIdentifier,
	inputArgumentInfosAddress := inputArgumentInfosAddress,
	inputArgumentInfosSize := inputArgumentInfosSize,
	inputConstantArgumentsAddress := inputConstantArgumentsAddress,
	inputConstantArgumentsSize := inputConstantArgumentsSize,
	inputDynamicArgumentsAddress := inputDynamicArgumentsAddress,
	inputDynamicArgumentsSize := inputDynamicArgumentsSize,
	outputArgumentInfosAddress := outputArgumentInfosAddress,
	outputArgumentInfosSize := outputArgumentInfosSize,
	outputArgumentsInfoAndDataAddress := outputArgumentsInfoAndDataAddress,
	outputArgumentsInfoAndDataSize := outputArgumentsInfoAndDataSize,
	numberOfReceivedBytesCount := numberOfReceivedBytesCount,
	operationTimeout := operationTimeout
);

AddMethodCallByNamespaceUri := _RequestItems.Append(requestItem);
END_METHOD

METHOD AddReadByNamespaceIndex : DINT
VAR_INPUT
	namespaceIndex : UINT;
	identifierType : Tc3_PLCopen_OpcUa.E_UAIdentifierType;
	identifier : STRING(Tc2_System.MAX_STRING_LENGTH);
	nodeAdditionalInfo : Tc3_PLCopen_OpcUa.ST_UANodeAdditionalInfo;
	targetVariable : ANY;
	receivedBytesCountTarget : POINTER TO UDINT;
	operationTimeout : TIME := T#0S;
END_VAR
VAR_OUTPUT
	exception : Exception;
END_VAR
VAR
	requestItem : POINTER TO OpcUaDAReadRequestItem;
END_VAR
AddReadByNamespaceIndex := -1;

IF Busy THEN
	ExceptionHelper.Throw(0, "OpcUaRequest is executing", __POUNAME(), ClassName, CurrentNamespace.Name, __POSITION());
	RETURN;
END_IF

_TimeoutTimer.Interval := _TimeoutTimer.Interval + operationTimeout;

requestItem := __NEW(OpcUaDAReadRequestItem);

requestItem^.Initialize(
	namespaceUri := '',
	namespaceIndex := namespaceIndex,
	identifierType := identifierType,
	identifier := identifier,
	nodeAdditionalInfo := nodeAdditionalInfo,
	targetVariable := targetVariable,
	numberOfReceivedBytesCount := receivedBytesCountTarget,
	operationTimeout := operationTimeout
);

AddReadByNamespaceIndex := _RequestItems.Append(requestItem);
END_METHOD

METHOD AddReadByNamespaceUri : DINT
VAR_INPUT
	namespaceUri : STRING(Tc2_System.MAX_STRING_LENGTH);
	identifierType : Tc3_PLCopen_OpcUa.E_UAIdentifierType;
	identifier : STRING(Tc2_System.MAX_STRING_LENGTH);
	nodeAdditionalInfo : Tc3_PLCopen_OpcUa.ST_UANodeAdditionalInfo;
	targetVariable : ANY;
	receivedBytesCountTarget : POINTER TO UDINT;
	operationTimeout : TIME := T#0S;
END_VAR
VAR_OUTPUT
	exception : Exception;
END_VAR
VAR
	namespaceUriPointer : POINTER TO STRING(MAX_STRING_LENGTH);
	getNamespaceIndex : POINTER TO Tc3_PLCopen_OpcUa.UA_GetNamespaceIndex;
	requestItem : POINTER TO OpcUaDAReadRequestItem;
END_VAR
AddReadByNamespaceUri := -1;

IF Busy THEN
	ExceptionHelper.Throw(0, "OpcUaRequest is executing", __POUNAME(), ClassName, CurrentNamespace.Name, __POSITION());
	RETURN;
END_IF

IF namespaceUri = '' THEN
	ExceptionHelper.Throw(0, "Parameter 'namespaceUri' is empty", __POUNAME(), ClassName, CurrentNamespace.Name, __POSITION());
	RETURN;	
END_IF

_TimeoutTimer.Interval := _TimeoutTimer.Interval + operationTimeout;

// try get existing namespace index request
getNamespaceIndex := _NamespaceUris.GetValueByKey(ADR(namespaceUri));

IF getNamespaceIndex <> 0 THEN
	IF operationTimeout > getNamespaceIndex^.Timeout THEN
		getNamespaceIndex^.Timeout := operationTimeout;	
	END_IF
// if not exists then create new request
ELSE
	namespaceUriPointer := __NEW(STRING(MAX_STRING_LENGTH));
	namespaceUriPointer^ := namespaceUri;
	
	getNamespaceIndex := __NEW(Tc3_PLCopen_OpcUa.UA_GetNamespaceIndex);
	getNamespaceIndex^.NamespaceUri := namespaceUri;
	getNamespaceIndex^.Timeout := operationTimeout;	
	
	_NamespaceUris.Set(namespaceUriPointer, getNamespaceIndex, TRUE, TRUE);
END_IF

requestItem := __NEW(OpcUaDAReadRequestItem);

requestItem^.Initialize(
	namespaceUri := namespaceUri,
	namespaceIndex := 0,
	identifierType := identifierType,
	identifier := identifier,
	nodeAdditionalInfo := nodeAdditionalInfo,
	targetVariable := targetVariable,
	numberOfReceivedBytesCount := receivedBytesCountTarget,
	operationTimeout := operationTimeout
);

AddReadByNamespaceUri := _RequestItems.Append(requestItem);
END_METHOD

METHOD AddWriteByNamespaceIndex : DINT
VAR_INPUT
	namespaceIndex : UINT;
	identifierType : Tc3_PLCopen_OpcUa.E_UAIdentifierType;
	identifier : STRING(Tc2_System.MAX_STRING_LENGTH);
	nodeAdditionalInfo : Tc3_PLCopen_OpcUa.ST_UANodeAdditionalInfo;
	sourceVariable : ANY;
	operationTimeout : TIME := T#0S;
END_VAR
VAR_OUTPUT
	exception : Exception;
END_VAR
VAR
	requestItem : POINTER TO OpcUaDAWriteRequestItem;
END_VAR
AddWriteByNamespaceIndex := -1;

IF Busy THEN
	ExceptionHelper.Throw(0, "OpcUaRequest is executing", __POUNAME(), ClassName, CurrentNamespace.Name, __POSITION());
	RETURN;
END_IF

_TimeoutTimer.Interval := _TimeoutTimer.Interval + operationTimeout;

requestItem := __NEW(OpcUaDAWriteRequestItem);

requestItem^.Initialize(
	namespaceUri := '',
	namespaceIndex := namespaceIndex,
	identifierType := identifierType,
	identifier := identifier,
	nodeAdditionalInfo := nodeAdditionalInfo,
	sourceVariable := sourceVariable,
	operationTimeout := operationTimeout
);

AddWriteByNamespaceIndex := _RequestItems.Append(requestItem);
END_METHOD

METHOD AddWriteByNamespaceUri : DINT
VAR_INPUT
	namespaceUri : STRING(Tc2_System.MAX_STRING_LENGTH);
	identifierType : Tc3_PLCopen_OpcUa.E_UAIdentifierType;
	identifier : STRING(Tc2_System.MAX_STRING_LENGTH);
	nodeAdditionalInfo : Tc3_PLCopen_OpcUa.ST_UANodeAdditionalInfo;
	sourceVariable : ANY;
	operationTimeout : TIME := T#0S;
END_VAR
VAR_OUTPUT
	exception : Exception;
END_VAR
VAR
	namespaceUriPointer : POINTER TO STRING(MAX_STRING_LENGTH);
	getNamespaceIndex : POINTER TO Tc3_PLCopen_OpcUa.UA_GetNamespaceIndex;
	requestItem : POINTER TO OpcUaDAWriteRequestItem;
END_VAR
AddWriteByNamespaceUri := -1;

IF Busy THEN
	ExceptionHelper.Throw(0, "OpcUaRequest is executing", __POUNAME(), ClassName, CurrentNamespace.Name, __POSITION());
	RETURN;
END_IF

IF namespaceUri = '' THEN
	ExceptionHelper.Throw(0, "Parameter 'namespaceUri' is empty", __POUNAME(), ClassName, CurrentNamespace.Name, __POSITION());
	RETURN;	
END_IF

_TimeoutTimer.Interval := _TimeoutTimer.Interval + operationTimeout;

// try get existing namespace index request
getNamespaceIndex := _NamespaceUris.GetValueByKey(ADR(namespaceUri));

IF getNamespaceIndex <> 0 THEN
	IF operationTimeout > getNamespaceIndex^.Timeout THEN
		getNamespaceIndex^.Timeout := operationTimeout;	
	END_IF
// if not exists then create new request
ELSE
	namespaceUriPointer := __NEW(STRING(MAX_STRING_LENGTH));
	namespaceUriPointer^ := namespaceUri;
	
	getNamespaceIndex := __NEW(Tc3_PLCopen_OpcUa.UA_GetNamespaceIndex);
	getNamespaceIndex^.NamespaceUri := namespaceUri;
	getNamespaceIndex^.Timeout := operationTimeout;	
	
	_NamespaceUris.Set(namespaceUriPointer, getNamespaceIndex, TRUE, TRUE);
END_IF

requestItem := __NEW(OpcUaDAWriteRequestItem);

requestItem^.Initialize(
	namespaceUri := namespaceUri,
	namespaceIndex := 0,
	identifierType := identifierType,
	identifier := identifier,
	nodeAdditionalInfo := nodeAdditionalInfo,
	sourceVariable := sourceVariable,
	operationTimeout := operationTimeout
);

AddWriteByNamespaceUri := _RequestItems.Append(requestItem);
END_METHOD

{attribute 'monitoring' := 'call'}
{attribute 'OPC.UA.DA' := '1'}
{attribute 'OPC.UA.DA.Property' := '1'}
PROPERTY Busy : BOOL
GET
Busy := _State <> OPC_UA_COMMUNICATOR_STATE.IDLE;
END_GET
END_PROPERTY

{attribute 'monitoring' := 'call'}
PROPERTY ClassName : STRING
GET
ClassName := _ClassName;
END_GET
END_PROPERTY

METHOD PRIVATE closeConnection : OPC_UA_ACTION_EXECUTION_STATE
_Connect(Execute := FALSE);
_Disconnect(Execute := TRUE, ConnectionHdl := _Connect.ConnectionHdl);

IF _Disconnect.Error THEN	
	IF _LastException.Empty THEN
		_LastExceptionHelper.Throw(_Disconnect.ErrorID, WCONCAT("UA_Disconnect error ", TO_WSTRING(_Disconnect.ErrorID)), __POUNAME(), ClassName, CurrentNamespace.Name, __POSITION());
	END_IF
 
	closeConnection := OPC_UA_ACTION_EXECUTION_STATE.ERROR;
ELSIF _Disconnect.Done THEN
	closeConnection := OPC_UA_ACTION_EXECUTION_STATE.DONE;
ELSE
	closeConnection := OPC_UA_ACTION_EXECUTION_STATE.BUSY;
END_IF
END_METHOD

PROPERTY CommunicationTypeName : STRING
GET
CommunicationTypeName := 'OPC-UA';
END_GET
END_PROPERTY

{attribute 'monitoring' := 'call'}
{attribute 'OPC.UA.DA' := '1'}
{attribute 'OPC.UA.DA.Property' := '1'}
PROPERTY DataProcessed : BOOL
GET
DataProcessed := _DataProcessed;
END_GET
END_PROPERTY

{attribute 'monitoring' := 'call'}
{attribute 'OPC.UA.DA' := '1'}
{attribute 'OPC.UA.DA.Property' := '1'}
PROPERTY Error : BOOL
GET
Error := _State = OPC_UA_COMMUNICATOR_STATE.IDLE AND_THEN NOT _LastException.Empty;
END_GET
END_PROPERTY

METHOD Execute
VAR
	prevState : OPC_UA_COMMUNICATOR_STATE;
END_VAR
VAR
	actionState : OPC_UA_ACTION_EXECUTION_STATE;
END_VAR
prevState := _State;
_DataProcessed := FALSE;
_OperationTimer.Execute();

StateMachine:

// state machine logic
CASE _State OF
	OPC_UA_COMMUNICATOR_STATE.CONNECT:
		actionState := openConnection();
		
		CASE actionState OF
			OPC_UA_ACTION_EXECUTION_STATE.DONE:
				_State := OPC_UA_COMMUNICATOR_STATE.GET_NAMESPACE_INDEX;
				JMP StateMachine;
			
			OPC_UA_ACTION_EXECUTION_STATE.ERROR:
				_State := OPC_UA_COMMUNICATOR_STATE.IDLE;
				RETURN;
		END_CASE
	
	OPC_UA_COMMUNICATOR_STATE.GET_NAMESPACE_INDEX:
		actionState := getNamespaceIndex();
		
		CASE actionState OF
			OPC_UA_ACTION_EXECUTION_STATE.DONE:
				_State := OPC_UA_COMMUNICATOR_STATE.GET_NODE_HANDLE;
				JMP StateMachine;
			
			OPC_UA_ACTION_EXECUTION_STATE.ERROR:
				_State := OPC_UA_COMMUNICATOR_STATE.DISCONNECT;
				JMP StateMachine;
		END_CASE	
		
	OPC_UA_COMMUNICATOR_STATE.GET_NODE_HANDLE:
		actionState := getNodeHandle();
		
		CASE actionState OF
			OPC_UA_ACTION_EXECUTION_STATE.DONE:
				_State := OPC_UA_COMMUNICATOR_STATE.PERFORM_ACTION;
				_OperationTimer.Start();
				JMP StateMachine;
			
			OPC_UA_ACTION_EXECUTION_STATE.ERROR:
				_State := OPC_UA_COMMUNICATOR_STATE.DISCONNECT;
				JMP StateMachine;
		END_CASE
	
	OPC_UA_COMMUNICATOR_STATE.PERFORM_ACTION:
		actionState := performAction();
		
		CASE actionState OF
			OPC_UA_ACTION_EXECUTION_STATE.DONE:
				_DataProcessed := TRUE;	
				CycleCount := CycleCount + 1;
				
				IF CyclicMode THEN
					_State := OPC_UA_COMMUNICATOR_STATE.WAIT_FOR_NEXT_CYCLE;			
					JMP StateMachine;			
				ELSE	
					_State := OPC_UA_COMMUNICATOR_STATE.RELEASE_NODE_HANDLE;		
				END_IF
			
			OPC_UA_ACTION_EXECUTION_STATE.ERROR:
				_State := OPC_UA_COMMUNICATOR_STATE.RELEASE_NODE_HANDLE;
				JMP StateMachine;
		END_CASE	

	OPC_UA_COMMUNICATOR_STATE.WAIT_FOR_NEXT_CYCLE:
		IF NOT _DataProcessed AND_THEN _OperationTimer.Interval >= CycleInterval THEN	
			resetAction();
			_State := OPC_UA_COMMUNICATOR_STATE.PERFORM_ACTION;				
			_OperationTimer.Start();
			JMP StateMachine;	
		END_IF	
	
	OPC_UA_COMMUNICATOR_STATE.RELEASE_NODE_HANDLE:
		actionState := releaseNodeHandle();
		
		CASE actionState OF
			OPC_UA_ACTION_EXECUTION_STATE.DONE, OPC_UA_ACTION_EXECUTION_STATE.ERROR:
				_State := OPC_UA_COMMUNICATOR_STATE.DISCONNECT;
				JMP StateMachine;
		END_CASE	
	
	OPC_UA_COMMUNICATOR_STATE.DISCONNECT:
		actionState := closeConnection();
		
		IF actionState = OPC_UA_ACTION_EXECUTION_STATE.DONE OR_ELSE actionState = OPC_UA_ACTION_EXECUTION_STATE.ERROR THEN
			_State := OPC_UA_COMMUNICATOR_STATE.IDLE;			
		END_IF
END_CASE

// check operation timeout (except for connect and disconnect)
IF Busy 
	AND_THEN _State <> OPC_UA_COMMUNICATOR_STATE.CONNECT 
	AND_THEN _State <> OPC_UA_COMMUNICATOR_STATE.DISCONNECT 
	AND_THEN _State <> OPC_UA_COMMUNICATOR_STATE.WAIT_FOR_NEXT_CYCLE 
THEN
	IF prevState <> _State THEN
		_TimeoutTimer.Start();
	ELSE
		_TimeoutTimer.Execute();
		
		IF _TimeoutTimer.Done THEN			
			IF _LastException.Empty THEN
				_LastExceptionHelper.Throw(1817, WCONCAT("Operation timeout in state ", TO_WSTRING(_State)), __POUNAME(), ClassName, CurrentNamespace.Name, __POSITION());
			END_IF
			
			CASE _State OF
				OPC_UA_COMMUNICATOR_STATE.GET_NAMESPACE_INDEX:
					_State := OPC_UA_COMMUNICATOR_STATE.DISCONNECT;
				
				OPC_UA_COMMUNICATOR_STATE.GET_NODE_HANDLE:
					_State := OPC_UA_COMMUNICATOR_STATE.DISCONNECT;
				
				OPC_UA_COMMUNICATOR_STATE.PERFORM_ACTION:
					_State := OPC_UA_COMMUNICATOR_STATE.RELEASE_NODE_HANDLE;
					
				OPC_UA_COMMUNICATOR_STATE.RELEASE_NODE_HANDLE:
					_State := OPC_UA_COMMUNICATOR_STATE.DISCONNECT;
			END_CASE			
		END_IF
	END_IF	
END_IF
END_METHOD

METHOD FB_exit : BOOL
VAR_INPUT
	bInCopyCode : BOOL; // if TRUE, the exit method is called for exiting an instance that is copied afterwards (online change).
END_VAR
_NamespaceUris.Clear(TRUE, TRUE);
_RequestItems.Clear(TRUE);
END_METHOD

METHOD getNamespaceIndex : OPC_UA_ACTION_EXECUTION_STATE
VAR
	i, j : DINT;
	functionBlock : POINTER TO Tc3_PLCopen_OpcUa.UA_GetNamespaceIndex;
	request : POINTER TO OpcUaDARequestItem;
END_VAR
getNamespaceIndex := OPC_UA_ACTION_EXECUTION_STATE.DONE;

FOR i := 0 TO _NamespaceUris.Count - 1 DO
	functionBlock := _NamespaceUris.GetValueByIndex(i);
	
	functionBlock^(Execute := TRUE, ConnectionHdl := _Connect.ConnectionHdl);

	IF functionBlock^.Error THEN
		IF getNamespaceIndex <> OPC_UA_ACTION_EXECUTION_STATE.ERROR THEN		
			IF _LastException.Empty THEN
				_LastExceptionHelper.Throw(functionBlock^.ErrorID, WStringHelper.Concat5("UA_GetNamespaceIndex error ", TO_WSTRING(functionBlock^.ErrorID), " (NamespaceUri = '", TO_WSTRING(functionBlock^.NamespaceUri), "')"), __POUNAME(), ClassName, CurrentNamespace.Name, __POSITION());				
			END_IF
		
			getNamespaceIndex := OPC_UA_ACTION_EXECUTION_STATE.ERROR;			
		END_IF
		
		AdsLogger.LogMessage(LOGGING_LEVEL.INFORMATION, WStringHelper.Concat3("---OpcUaRequest getNamespaceIndex error: ", "UA_GetNamespaceIndex error ", TO_WSTRING(functionBlock^.ErrorID)));
	ELSIF functionBlock^.Done THEN
		FOR j := 0 TO _RequestItems.Count - 1 DO
			request := _RequestItems.Get(j);
			request^.SetNamespaceIndexForNamespaceUri(functionBlock^.NamespaceUri, functionBlock^.NamespaceIndex);
		END_FOR
	ELSE
		IF getNamespaceIndex <> OPC_UA_ACTION_EXECUTION_STATE.ERROR THEN
			getNamespaceIndex := OPC_UA_ACTION_EXECUTION_STATE.BUSY;			
		END_IF			
	END_IF
END_FOR

IF getNamespaceIndex = OPC_UA_ACTION_EXECUTION_STATE.DONE THEN
	AdsLogger.LogMessage(LOGGING_LEVEL.INFORMATION, "---OpcUaRequest getNamespaceIndex done");	
END_IF
END_METHOD

METHOD getNodeHandle : OPC_UA_ACTION_EXECUTION_STATE
VAR
	i : DINT;
	requestItem : POINTER TO OpcUaRequestItem;
	requestItemState : OPC_UA_ACTION_EXECUTION_STATE;	
	exception : Exception;
END_VAR
getNodeHandle := OPC_UA_ACTION_EXECUTION_STATE.DONE;

FOR i := 0 TO _RequestItems.Count - 1 DO
	requestItem := _RequestItems.Get(i);
	
	requestItemState := requestItem^.GetHandle(_Connect.ConnectionHdl, exception => exception);
	
	CASE requestItemState OF
		OPC_UA_ACTION_EXECUTION_STATE.BUSY:
			IF getNodeHandle <> OPC_UA_ACTION_EXECUTION_STATE.ERROR THEN
				getNodeHandle := OPC_UA_ACTION_EXECUTION_STATE.BUSY;			
			END_IF
							
		OPC_UA_ACTION_EXECUTION_STATE.ERROR:
			IF getNodeHandle <> OPC_UA_ACTION_EXECUTION_STATE.ERROR THEN
				IF _LastException.Empty THEN
					_LastException := exception;				
				END_IF
				
				getNodeHandle := OPC_UA_ACTION_EXECUTION_STATE.ERROR;							
			END_IF
	END_CASE
END_FOR

IF getNodeHandle = OPC_UA_ACTION_EXECUTION_STATE.DONE THEN
	AdsLogger.LogMessage(LOGGING_LEVEL.INFORMATION, "---OpcUaRequest getNodeHandle done");
END_IF
END_METHOD

METHOD PROTECTED InternalClear : BOOL
VAR_OUTPUT
	exception : Exception;
END_VAR
_NamespaceUris.Clear(TRUE, TRUE);
_RequestItems.Clear(TRUE);

InternalClear := TRUE;
END_METHOD

METHOD PROTECTED InternalConfigure : BOOL
VAR_INPUT
	settings : REFERENCE TO CommunicationSettings;
END_VAR
VAR_OUTPUT
	exception : Exception;
END_VAR
VAR
	opcUaSettings : POINTER TO OpcUaCommunicationSettings;
END_VAR
opcUaSettings := ADR(settings);

IF opcUaSettings^.ServerUrl = '' THEN
	ExceptionHelper.Throw(0, "settings.ServerUrl is empty", __POUNAME(), ClassName, CurrentNamespace.Name, __POSITION());
	RETURN;	
END_IF

_Connect.ServerUrl := opcUaSettings^.ServerUrl;
_Connect.SessionConnectInfo := opcUaSettings^.SessionConnectInfo;
_Connect.Timeout := opcUaSettings^.ConnectionTimeout;
_Disconnect.Timeout := opcUaSettings^.ConnectionTimeout;

_TimeoutTimer.Interval := opcUaSettings^.ConnectionTimeout;

InternalConfigure := TRUE;
END_METHOD

METHOD PROTECTED InternalStart : BOOL
VAR_OUTPUT
	exception : Exception;
END_VAR
VAR
	i : DINT;
	requestItem : POINTER TO OpcUaRequestItem;
	getNamespaceIndex : POINTER TO Tc3_PLCopen_OpcUa.UA_GetNamespaceIndex;
END_VAR
_State := OPC_UA_COMMUNICATOR_STATE.CONNECT;

_OperationTimer.Interval := T#1H;

_Connect(Execute := FALSE);

FOR i := 0 TO _NamespaceUris.Count - 1 DO
	getNamespaceIndex := _NamespaceUris.GetValueByIndex(i);
	
	getNamespaceIndex^(Execute := FALSE);
END_FOR

FOR i := 0 TO _RequestItems.Count - 1 DO
	requestItem := _RequestItems.Get(i);	
	requestItem^.Reset();
END_FOR

_TimeoutTimer.Start();

InternalStart := TRUE;
END_METHOD

METHOD PROTECTED InternalStop
CASE _State OF
	OPC_UA_COMMUNICATOR_STATE.CONNECT, 
	OPC_UA_COMMUNICATOR_STATE.GET_NAMESPACE_INDEX,
	OPC_UA_COMMUNICATOR_STATE.GET_NODE_HANDLE:
		_State := OPC_UA_COMMUNICATOR_STATE.DISCONNECT;
			
	OPC_UA_COMMUNICATOR_STATE.PERFORM_ACTION,
	OPC_UA_COMMUNICATOR_STATE.WAIT_FOR_NEXT_CYCLE:
		_State := OPC_UA_COMMUNICATOR_STATE.RELEASE_NODE_HANDLE;
	
	OPC_UA_COMMUNICATOR_STATE.RELEASE_NODE_HANDLE:
		_State := OPC_UA_COMMUNICATOR_STATE.DISCONNECT;

	//OPC_UA_SINGLE_REQUEST_STATE.DISCONNECT:		
END_CASE

_OperationTimer.Stop();
END_METHOD

METHOD PRIVATE openConnection : OPC_UA_ACTION_EXECUTION_STATE
_Disconnect(Execute := FALSE);
_Connect(Execute := TRUE);

IF _Connect.Error THEN
	LastExceptionHelper.Throw(_Connect.ErrorID, WStringHelper.Concat5("UA_Connect error ", TO_WSTRING(_Connect.ErrorID), " (ServerUrl = '", TO_WSTRING(_Connect.ServerUrl), "')"), __POUNAME(), ClassName, CurrentNamespace.Name, __POSITION());			
	openConnection := OPC_UA_ACTION_EXECUTION_STATE.ERROR;
ELSIF _Connect.Done THEN
	openConnection := OPC_UA_ACTION_EXECUTION_STATE.DONE;
ELSE
	openConnection := OPC_UA_ACTION_EXECUTION_STATE.BUSY;
END_IF
END_METHOD

METHOD performAction : OPC_UA_ACTION_EXECUTION_STATE
VAR
	i : DINT;
	requestItem : POINTER TO OpcUaRequestItem;
	requestItemState : OPC_UA_ACTION_EXECUTION_STATE;	
	exception : Exception;
END_VAR
performAction := OPC_UA_ACTION_EXECUTION_STATE.DONE;

FOR i := 0 TO _RequestItems.Count - 1 DO
	requestItem := _RequestItems.Get(i);
	
	requestItemState := requestItem^.PerformAction(exception => exception);
	
	CASE requestItemState OF
		OPC_UA_ACTION_EXECUTION_STATE.BUSY:
			IF performAction <> OPC_UA_ACTION_EXECUTION_STATE.ERROR THEN
				performAction := OPC_UA_ACTION_EXECUTION_STATE.BUSY;			
			END_IF
							
		OPC_UA_ACTION_EXECUTION_STATE.ERROR:
			IF performAction <> OPC_UA_ACTION_EXECUTION_STATE.ERROR THEN
				IF _LastException.Empty THEN
					_LastException := exception;				
				END_IF
				
				performAction := OPC_UA_ACTION_EXECUTION_STATE.ERROR;							
			END_IF
	END_CASE
END_FOR

IF performAction = OPC_UA_ACTION_EXECUTION_STATE.DONE THEN
	AdsLogger.LogMessage(LOGGING_LEVEL.INFORMATION, "---OpcUaRequest performAction done");
END_IF
END_METHOD

METHOD releaseNodeHandle : OPC_UA_ACTION_EXECUTION_STATE
VAR
	i : DINT;
	requestItem : POINTER TO OpcUaRequestItem;
	requestItemState : OPC_UA_ACTION_EXECUTION_STATE;	
	exception : Exception;
END_VAR
releaseNodeHandle := OPC_UA_ACTION_EXECUTION_STATE.DONE;

FOR i := 0 TO _RequestItems.Count - 1 DO
	requestItem := _RequestItems.Get(i);
	
	requestItemState := requestItem^.ReleaseHandle(exception => exception);
	
	CASE requestItemState OF
		OPC_UA_ACTION_EXECUTION_STATE.BUSY:
			IF releaseNodeHandle <> OPC_UA_ACTION_EXECUTION_STATE.ERROR THEN
				releaseNodeHandle := OPC_UA_ACTION_EXECUTION_STATE.BUSY;			
			END_IF
							
		OPC_UA_ACTION_EXECUTION_STATE.ERROR:
			IF releaseNodeHandle <> OPC_UA_ACTION_EXECUTION_STATE.ERROR THEN
				IF _LastException.Empty THEN
					_LastException := exception;				
				END_IF
				
				releaseNodeHandle := OPC_UA_ACTION_EXECUTION_STATE.ERROR;							
			END_IF
	END_CASE
END_FOR

IF releaseNodeHandle = OPC_UA_ACTION_EXECUTION_STATE.DONE THEN
	AdsLogger.LogMessage(LOGGING_LEVEL.INFORMATION, "---OpcUaRequest releaseNodeHandle done");
END_IF
END_METHOD

METHOD resetAction
VAR
	i : DINT;
	requestItem : POINTER TO OpcUaRequestItem;
END_VAR
FOR i := 0 TO _RequestItems.Count - 1 DO
	requestItem := _RequestItems.Get(i);
	requestItem^.ResetAction();
END_FOR
END_METHOD

PROPERTY VariablesCount : DINT
GET
VariablesCount := _RequestItems.Count;
END_GET
END_PROPERTY

END_FUNCTION_BLOCK

// ---- Communication/OPC_UA/RequestItems/OpcUaMethodCallRequestItem.TcPOU
{attribute 'enable_dynamic_creation'}	
FUNCTION_BLOCK OpcUaMethodCallRequestItem EXTENDS OpcUaRequestItem
VAR
	_ClassName : STRING := __POUNAME();

	_ObjectNamespaceUri : STRING(Tc2_System.MAX_STRING_LENGTH);
	_ObjectNodeId: Tc3_PLCopen_OpcUa.ST_UANodeID;		
	_ObjectNamespaceIndexValid : BOOL;

	_MethodNamespaceUri : STRING(Tc2_System.MAX_STRING_LENGTH);
	_MethodNodeId: Tc3_PLCopen_OpcUa.ST_UANodeID;		
	_MethodNamespaceIndexValid : BOOL;

	_NumberOfReceivedBytesCount : POINTER TO UDINT;
	
	_GetMethodHandle : Tc3_PLCopen_OpcUa.UA_MethodGetHandle;
	_MethodCall : Tc3_PLCopen_OpcUa.UA_MethodCall;
	_ReleaseMethodHandle : Tc3_PLCopen_OpcUa.UA_MethodReleaseHandle;	
END_VAR

{attribute 'monitoring' := 'call'}
PROPERTY ClassName : STRING
GET
ClassName := _ClassName;
END_GET
END_PROPERTY

METHOD GetHandle : OPC_UA_ACTION_EXECUTION_STATE
VAR_INPUT
	connectionHandle : DWORD;
END_VAR
VAR_OUTPUT
	exception : Exception;
END_VAR
_ConnectionHandle := connectionHandle;

GetHandle := OPC_UA_ACTION_EXECUTION_STATE.DONE;
	
IF NOT _ObjectNamespaceIndexValid THEN
	ExceptionHelper.Throw(0, WStringHelper.Concat3("UA__GetMethodHandle error: invalid object namespace index for namespace '", TO_WSTRING(_ObjectNamespaceUri), "'"), __POUNAME(), ClassName, CurrentNamespace.Name, __POSITION());				
	GetHandle := OPC_UA_ACTION_EXECUTION_STATE.ERROR;				
	AdsLogger.LogMessage(LOGGING_LEVEL.INFORMATION, WStringHelper.Concat3("---OpcUaRequest GetNodeHandle error: invalid object namespace index for namespace '", TO_WSTRING(_ObjectNamespaceUri), "'"));
ELSIF NOT _MethodNamespaceIndexValid THEN
	ExceptionHelper.Throw(0, WStringHelper.Concat3("UA__GetMethodHandle error: invalid method namespace index for namespace '", TO_WSTRING(_MethodNamespaceUri), "'"), __POUNAME(), ClassName, CurrentNamespace.Name, __POSITION());				
	GetHandle := OPC_UA_ACTION_EXECUTION_STATE.ERROR;				
	AdsLogger.LogMessage(LOGGING_LEVEL.INFORMATION, WStringHelper.Concat3("---OpcUaRequest GetMethodHandle error: invalid method namespace index for namespace '", TO_WSTRING(_MethodNamespaceUri), "'"));
ELSE
	_GetMethodHandle(Execute := TRUE, ConnectionHdl := _ConnectionHandle, ObjectNodeID := _ObjectNodeId, MethodNodeID := _MethodNodeId);

	IF _GetMethodHandle.Error THEN
		ExceptionHelper.Throw(_GetMethodHandle.ErrorID, WStringHelper.Concat7("UA_GetMethodHandle error ", TO_WSTRING(_GetMethodHandle.ErrorID), " (ObjectNodeID='", TO_WSTRING(_ObjectNodeId.sIdentifier), "', MethodNodeID='", TO_WSTRING(_MethodNodeId.sIdentifier), "')"), __POUNAME(), ClassName, CurrentNamespace.Name, __POSITION());					
		GetHandle := OPC_UA_ACTION_EXECUTION_STATE.ERROR;					
		AdsLogger.LogMessage(LOGGING_LEVEL.INFORMATION, WStringHelper.Concat3("---OpcUaRequest GetMethodHandle error: ", "UA_GetMethodHandle error ", TO_WSTRING(_GetMethodHandle.ErrorID)));
	ELSIF _GetMethodHandle.Busy THEN
		GetHandle := OPC_UA_ACTION_EXECUTION_STATE.BUSY;			
	END_IF
END_IF
END_METHOD

METHOD Initialize
VAR_INPUT
	objectNamespaceUri : STRING(Tc2_System.MAX_STRING_LENGTH); // empty string if index used
	objectNamespaceIndex : UINT; // zero if namespace uri used
	objectIdentifierType : Tc3_PLCopen_OpcUa.E_UAIdentifierType;
	objectIdentifier : STRING(Tc2_System.MAX_STRING_LENGTH);	
	methodNamespaceUri : STRING(Tc2_System.MAX_STRING_LENGTH); // empty string if index used
	methodNamespaceIndex : UINT; // zero if namespace uri used
	methodIdentifierType : Tc3_PLCopen_OpcUa.E_UAIdentifierType;
	methodIdentifier : STRING(Tc2_System.MAX_STRING_LENGTH);
	inputArgumentInfosAddress : POINTER TO ST_UAMethodArgInfo;
	inputArgumentInfosSize : UDINT;
	inputConstantArgumentsAddress : PVOID;
	inputConstantArgumentsSize : UDINT;
	inputDynamicArgumentsAddress : PVOID;
	inputDynamicArgumentsSize : UDINT;
	outputArgumentInfosAddress : POINTER TO ST_UAMethodArgInfo;
	outputArgumentInfosSize : UDINT;
	outputArgumentsInfoAndDataAddress : POINTER TO OPC_UA_OUTPUT_ARGUMENT_INFO_AND_DATA;
	outputArgumentsInfoAndDataSize : UDINT;
	numberOfReceivedBytesCount : POINTER TO UDINT;
	operationTimeout : TIME := Tc2_System.DEFAULT_ADS_TIMEOUT;
END_VAR
IF objectNamespaceUri <> '' THEN
	_ObjectNamespaceUri := objectNamespaceUri;
	_ObjectNodeId.nNamespaceIndex := 0;
	_ObjectNamespaceIndexValid := FALSE;
ELSE
	_ObjectNamespaceUri := '';
	_ObjectNodeId.nNamespaceIndex := objectNamespaceIndex;
	_ObjectNamespaceIndexValid := TRUE;
END_IF

_ObjectNodeId.eIdentifierType := objectIdentifierType;
_ObjectNodeId.sIdentifier := objectIdentifier;

IF methodNamespaceUri <> '' THEN
	_MethodNamespaceUri := methodNamespaceUri;
	_MethodNodeId.nNamespaceIndex := 0;
	_MethodNamespaceIndexValid := FALSE;
ELSE
	_MethodNamespaceUri := '';
	_MethodNodeId.nNamespaceIndex := methodNamespaceIndex;
	_MethodNamespaceIndexValid := TRUE;
END_IF

_MethodNodeId.eIdentifierType := methodIdentifierType;
_MethodNodeId.sIdentifier := methodIdentifier;
_MethodCall.nNumberOfInputArguments := inputArgumentInfosSize / SIZEOF(ST_UAMethodArgInfo);
_MethodCall.pInputArgInfo := inputArgumentInfosAddress;
_MethodCall.cbInputArgInfo := inputArgumentInfosSize;
_MethodCall.pInputArgData := inputConstantArgumentsAddress;
_MethodCall.cbInputArgData := inputConstantArgumentsSize;
_MethodCall.pInputWriteData := inputDynamicArgumentsAddress;
_MethodCall.cbInputWriteData := inputDynamicArgumentsSize;
_MethodCall.nNumberOfOutputArguments := outputArgumentInfosSize / SIZEOF(ST_UAMethodArgInfo);
_MethodCall.pOutputArgInfo := outputArgumentInfosAddress;
_MethodCall.cbOutputArgInfo := outputArgumentInfosSize;
_MethodCall.pOutputArgInfoAndData := outputArgumentsInfoAndDataAddress;
_MethodCall.cbOutputArgInfoAndData := outputArgumentsInfoAndDataSize;

_NumberOfReceivedBytesCount := numberOfReceivedBytesCount;

_GetMethodHandle.Timeout := operationTimeout;
_MethodCall.Timeout := operationTimeout;
_ReleaseMethodHandle.Timeout := operationTimeout;
END_METHOD

METHOD PerformAction : OPC_UA_ACTION_EXECUTION_STATE
VAR_OUTPUT
	exception : Exception;
END_VAR
PerformAction := OPC_UA_ACTION_EXECUTION_STATE.DONE;

_MethodCall(Execute := TRUE, ConnectionHdl := _ConnectionHandle, MethodHdl := _GetMethodHandle.MethodHdl);
		
IF _MethodCall.Error THEN
	ExceptionHelper.Throw(_GetMethodHandle.ErrorID, WStringHelper.Concat7("UA_MethodCall error ", TO_WSTRING(_MethodCall.ErrorID), " (ObjectNodeID='", TO_WSTRING(_ObjectNodeId.sIdentifier), "', MethodNodeID='", TO_WSTRING(_MethodNodeId.sIdentifier), "')"), __POUNAME(), ClassName, CurrentNamespace.Name, __POSITION());					
	PerformAction := OPC_UA_ACTION_EXECUTION_STATE.ERROR;			
	AdsLogger.LogMessage(LOGGING_LEVEL.INFORMATION, WStringHelper.Concat3("---OpcUaRequest PerformAction error: ", "UA_MethodCall error ", TO_WSTRING(_MethodCall.ErrorID)));
ELSIF _MethodCall.Busy THEN
	PerformAction := OPC_UA_ACTION_EXECUTION_STATE.BUSY;
ELSIF _GetMethodHandle.Done AND_THEN _NumberOfReceivedBytesCount <> 0 THEN
 	_NumberOfReceivedBytesCount^ := _MethodCall.cbRead_R;
END_IF
END_METHOD

METHOD ReleaseHandle : OPC_UA_ACTION_EXECUTION_STATE
VAR_OUTPUT
	exception : Exception;
END_VAR
ReleaseHandle := OPC_UA_ACTION_EXECUTION_STATE.DONE;
	
_ReleaseMethodHandle(Execute := TRUE, ConnectionHdl := _ConnectionHandle, MethodHdl := _GetMethodHandle.MethodHdl);

IF _ReleaseMethodHandle.Error THEN
	ExceptionHelper.Throw(_ReleaseMethodHandle.ErrorID, WCONCAT("UA_ReleaseMethodHandle error ", TO_WSTRING(_ReleaseMethodHandle.ErrorID)), __POUNAME(), ClassName, CurrentNamespace.Name, __POSITION());
	ReleaseHandle := OPC_UA_ACTION_EXECUTION_STATE.ERROR;			
	AdsLogger.LogMessage(LOGGING_LEVEL.INFORMATION, WStringHelper.Concat3("---OpcUaRequest ReleaseMethodHandle error: ", "UA_ReleaseMethodHandle error ", TO_WSTRING(_ReleaseMethodHandle.ErrorID)));
ELSIF _ReleaseMethodHandle.Busy THEN
	ReleaseHandle := OPC_UA_ACTION_EXECUTION_STATE.BUSY;			
END_IF
END_METHOD

METHOD Reset
_GetMethodHandle(Execute := FALSE);
ResetAction();
_ReleaseMethodHandle(Execute := FALSE);
END_METHOD

METHOD ResetAction
_MethodCall(Execute := FALSE);
END_METHOD

METHOD SetNamespaceIndexForNamespaceUri
VAR_INPUT
	namespaceUri : STRING(Tc2_System.MAX_STRING_LENGTH);
	namespaceIndex : UINT;
END_VAR
IF NOT _ObjectNamespaceIndexValid AND_THEN _ObjectNamespaceUri = namespaceUri THEN
	_ObjectNodeId.nNamespaceIndex := namespaceIndex;
	_ObjectNamespaceIndexValid := TRUE;					
END_IF

IF NOT _MethodNamespaceIndexValid AND_THEN _MethodNamespaceUri = namespaceUri THEN
	_MethodNodeId.nNamespaceIndex := namespaceIndex;
	_MethodNamespaceIndexValid := TRUE;					
END_IF
END_METHOD

END_FUNCTION_BLOCK

// ---- Communication/OPC_UA/RequestItems/OpcUaRequestItem.TcPOU
FUNCTION_BLOCK ABSTRACT OpcUaRequestItem EXTENDS TC.ToolkitObject
VAR
	_ConnectionHandle : DWORD;
END_VAR

METHOD ABSTRACT GetHandle : OPC_UA_ACTION_EXECUTION_STATE
VAR_INPUT
	connectionHandle : DWORD;
END_VAR
VAR_OUTPUT
	exception : Exception;
END_VAR
END_METHOD

METHOD ABSTRACT PerformAction : OPC_UA_ACTION_EXECUTION_STATE
VAR_OUTPUT
	exception : Exception;
END_VAR
END_METHOD

METHOD ABSTRACT ReleaseHandle : OPC_UA_ACTION_EXECUTION_STATE
VAR_OUTPUT
	exception : Exception;
END_VAR
END_METHOD

METHOD ABSTRACT Reset
END_METHOD

METHOD ABSTRACT ResetAction
END_METHOD

METHOD ABSTRACT SetNamespaceIndexForNamespaceUri
VAR_INPUT
	namespaceUri : STRING(Tc2_System.MAX_STRING_LENGTH);
	namespaceIndex : UINT;
END_VAR
END_METHOD

END_FUNCTION_BLOCK

// ---- Communication/OPC_UA/RequestItems/OpcUaDAReadRequestItem.TcPOU
{attribute 'enable_dynamic_creation'}	
FUNCTION_BLOCK OpcUaDAReadRequestItem EXTENDS OpcUaDARequestItem
VAR
	_ClassName : STRING := __POUNAME();

	_Read : Tc3_PLCopen_OpcUa.UA_Read;
	_NumberOfReceivedBytesCount : POINTER TO UDINT;
END_VAR

{attribute 'monitoring' := 'call'}
PROPERTY ClassName : STRING
GET
ClassName := _ClassName;
END_GET
END_PROPERTY

METHOD Initialize
VAR_INPUT
	namespaceUri : STRING(Tc2_System.MAX_STRING_LENGTH); // empty string if index used
	namespaceIndex : UINT; // zero if namespace uri used
	identifierType : Tc3_PLCopen_OpcUa.E_UAIdentifierType;
	identifier : STRING(Tc2_System.MAX_STRING_LENGTH);
	nodeAdditionalInfo : Tc3_PLCopen_OpcUa.ST_UANodeAdditionalInfo;
	targetVariable : __SYSTEM.AnyType;
	numberOfReceivedBytesCount : POINTER TO UDINT;
	operationTimeout : TIME := Tc2_System.DEFAULT_ADS_TIMEOUT;
END_VAR
IF namespaceUri <> '' THEN
	_NamespaceUri := namespaceUri;
	_NodeId.nNamespaceIndex := 0;
	_NamespaceIndexValid := FALSE;
ELSE
	_NamespaceUri := '';
	_NodeId.nNamespaceIndex := namespaceIndex;
	_NamespaceIndexValid := TRUE;
END_IF

_NodeId.eIdentifierType := identifierType;
_NodeId.sIdentifier := identifier;

_Read.stNodeAddInfo := nodeAdditionalInfo;
_Read.pVariable := targetVariable.pValue;
_Read.cbData := TO_UDINT(targetVariable.diSize);

_NumberOfReceivedBytesCount := numberOfReceivedBytesCount;

_GetNodeHandle.Timeout := operationTimeout;
_Read.Timeout := operationTimeout;
_ReleaseNodeHandle.Timeout := operationTimeout;
END_METHOD

METHOD PerformAction : OPC_UA_ACTION_EXECUTION_STATE
VAR_OUTPUT
	exception : Exception;
END_VAR
PerformAction := OPC_UA_ACTION_EXECUTION_STATE.DONE;

_Read(Execute := TRUE, ConnectionHdl := _ConnectionHandle, NodeHdl := _GetNodeHandle.NodeHdl);
		
IF _Read.Error THEN
	ExceptionHelper.Throw(_Read.ErrorID, WStringHelper.Concat5("UA_Read error ", TO_WSTRING(_Read.ErrorID), " (Node identifier = '", TO_WSTRING(_NodeId.sIdentifier), "')"), __POUNAME(), ClassName, CurrentNamespace.Name, __POSITION());					
	PerformAction := OPC_UA_ACTION_EXECUTION_STATE.ERROR;			
	AdsLogger.LogMessage(LOGGING_LEVEL.INFORMATION, WStringHelper.Concat3("---OpcUaRequest PerformAction error: ", "UA_Read error ", TO_WSTRING(_Read.ErrorID)));
ELSIF _Read.Busy THEN
	PerformAction := OPC_UA_ACTION_EXECUTION_STATE.BUSY;
ELSIF _Read.Done AND_THEN _NumberOfReceivedBytesCount <> 0 THEN
 	_NumberOfReceivedBytesCount^ := _Read.cbData_R;
END_IF
END_METHOD

METHOD ResetAction
_Read(Execute := FALSE);
END_METHOD

END_FUNCTION_BLOCK

// ---- Communication/OPC_UA/RequestItems/OpcUaDARequestItem.TcPOU
FUNCTION_BLOCK ABSTRACT OpcUaDARequestItem EXTENDS OpcUaRequestItem
VAR
	_NamespaceUri : STRING(Tc2_System.MAX_STRING_LENGTH);
	_NodeId: Tc3_PLCopen_OpcUa.ST_UANodeID;		
	_NamespaceIndexValid : BOOL;
	
	_GetNodeHandle : Tc3_PLCopen_OpcUa.UA_NodeGetHandle;
	_ReleaseNodeHandle : Tc3_PLCopen_OpcUa.UA_NodeReleaseHandle;	
END_VAR

METHOD GetHandle : OPC_UA_ACTION_EXECUTION_STATE
VAR_INPUT
	connectionHandle : DWORD;
END_VAR
VAR_OUTPUT
	exception : Exception;
END_VAR
_ConnectionHandle := connectionHandle;

GetHandle := OPC_UA_ACTION_EXECUTION_STATE.DONE;
	
IF NOT _NamespaceIndexValid THEN
	ExceptionHelper.Throw(0, WStringHelper.Concat3("UA_GetNodeHandle error: invalid namespace index for namespace '", TO_WSTRING(_NamespaceUri), "'"), __POUNAME(), ClassName, CurrentNamespace.Name, __POSITION());				
	GetHandle := OPC_UA_ACTION_EXECUTION_STATE.ERROR;				
	AdsLogger.LogMessage(LOGGING_LEVEL.INFORMATION, WStringHelper.Concat3("---OpcUaRequest GetNodeHandle error: invalid namespace index for namespace '", TO_WSTRING(_NamespaceUri), "'"));
ELSE
	_GetNodeHandle(Execute := TRUE, ConnectionHdl := _ConnectionHandle, NodeID := _NodeId);

	IF _GetNodeHandle.Error THEN
		ExceptionHelper.Throw(_GetNodeHandle.ErrorID, WStringHelper.Concat5("UA_GetNodeHandle error ", TO_WSTRING(_GetNodeHandle.ErrorID), " (NodeID.sIdentifier = '", TO_WSTRING(_GetNodeHandle.NodeID.sIdentifier), "')"), __POUNAME(), ClassName, CurrentNamespace.Name, __POSITION());					
		GetHandle := OPC_UA_ACTION_EXECUTION_STATE.ERROR;					
		AdsLogger.LogMessage(LOGGING_LEVEL.INFORMATION, WStringHelper.Concat3("---OpcUaRequest GetNodeHandle error: ", "UA_GetNodeHandle error ", TO_WSTRING(_GetNodeHandle.ErrorID)));
	ELSIF _GetNodeHandle.Busy THEN
		GetHandle := OPC_UA_ACTION_EXECUTION_STATE.BUSY;			
	END_IF
END_IF
END_METHOD

METHOD ReleaseHandle : OPC_UA_ACTION_EXECUTION_STATE
VAR_OUTPUT
	exception : Exception;
END_VAR
ReleaseHandle := OPC_UA_ACTION_EXECUTION_STATE.DONE;
	
_ReleaseNodeHandle(Execute := TRUE, ConnectionHdl := _ConnectionHandle, NodeHdl := _GetNodeHandle.NodeHdl);

IF _ReleaseNodeHandle.Error THEN
	ExceptionHelper.Throw(_ReleaseNodeHandle.ErrorID, WCONCAT("UA_ReleaseNodeHandle error ", TO_WSTRING(_ReleaseNodeHandle.ErrorID)), __POUNAME(), ClassName, CurrentNamespace.Name, __POSITION());
	ReleaseHandle := OPC_UA_ACTION_EXECUTION_STATE.ERROR;			
	AdsLogger.LogMessage(LOGGING_LEVEL.INFORMATION, WStringHelper.Concat3("---OpcUaRequest ReleaseNodeHandle error: ", "UA_ReleaseNodeHandle error ", TO_WSTRING(_ReleaseNodeHandle.ErrorID)));
ELSIF _GetNodeHandle.Busy THEN
	ReleaseHandle := OPC_UA_ACTION_EXECUTION_STATE.BUSY;			
END_IF
END_METHOD

METHOD Reset
_GetNodeHandle(Execute := FALSE);
ResetAction();
_ReleaseNodeHandle(Execute := FALSE);
END_METHOD

METHOD SetNamespaceIndexForNamespaceUri
VAR_INPUT
	namespaceUri : STRING(Tc2_System.MAX_STRING_LENGTH);
	namespaceIndex : UINT;
END_VAR
IF NOT _NamespaceIndexValid AND_THEN _NamespaceUri = namespaceUri THEN
	_NodeId.nNamespaceIndex := namespaceIndex;
	_NamespaceIndexValid := TRUE;					
END_IF
END_METHOD

END_FUNCTION_BLOCK

// ---- Communication/OPC_UA/RequestItems/OpcUaDAWriteRequestItem.TcPOU
{attribute 'enable_dynamic_creation'}	
FUNCTION_BLOCK OpcUaDAWriteRequestItem EXTENDS OpcUaDARequestItem
VAR
	_ClassName : STRING := __POUNAME();

	_Write : Tc3_PLCopen_OpcUa.UA_Write;
END_VAR

{attribute 'monitoring' := 'call'}
PROPERTY ClassName : STRING
GET
ClassName := _ClassName;
END_GET
END_PROPERTY

METHOD Initialize
VAR_INPUT
	namespaceUri : STRING(Tc2_System.MAX_STRING_LENGTH); // empty string if index used
	namespaceIndex : UINT; // zero if namespace uri used
	identifierType : Tc3_PLCopen_OpcUa.E_UAIdentifierType;
	identifier : STRING(Tc2_System.MAX_STRING_LENGTH);
	nodeAdditionalInfo : Tc3_PLCopen_OpcUa.ST_UANodeAdditionalInfo;
	sourceVariable : __SYSTEM.AnyType;
	operationTimeout : TIME := Tc2_System.DEFAULT_ADS_TIMEOUT;
END_VAR
IF namespaceUri <> '' THEN
	_NamespaceUri := namespaceUri;
	_NodeId.nNamespaceIndex := 0;
	_NamespaceIndexValid := FALSE;
ELSE
	_NamespaceUri := '';
	_NodeId.nNamespaceIndex := namespaceIndex;
	_NamespaceIndexValid := TRUE;
END_IF

_NodeId.eIdentifierType := identifierType;
_NodeId.sIdentifier := identifier;

_Write.stNodeAddInfo := nodeAdditionalInfo;
_Write.pVariable := sourceVariable.pValue;
_Write.cbData := TO_UDINT(sourceVariable.diSize);

_GetNodeHandle.Timeout := operationTimeout;
_Write.Timeout := operationTimeout;
_ReleaseNodeHandle.Timeout := operationTimeout;
END_METHOD

METHOD PerformAction : OPC_UA_ACTION_EXECUTION_STATE
VAR_OUTPUT
	exception : Exception;
END_VAR
PerformAction := OPC_UA_ACTION_EXECUTION_STATE.DONE;
	
_Write(Execute := TRUE, ConnectionHdl := _ConnectionHandle, NodeHdl := _GetNodeHandle.NodeHdl);
		
IF _Write.Error THEN
	ExceptionHelper.Throw(_Write.ErrorID, WStringHelper.Concat5("UA_Write error ", TO_WSTRING(_Write.ErrorID), " (Node identifier = '", TO_WSTRING(_NodeId.sIdentifier), "')"), __POUNAME(), ClassName, CurrentNamespace.Name, __POSITION());;					
	PerformAction := OPC_UA_ACTION_EXECUTION_STATE.ERROR;				
	AdsLogger.LogMessage(LOGGING_LEVEL.INFORMATION, WStringHelper.Concat3("---OpcUaRequest performAction error: ", "UA_Write error ", TO_WSTRING(_Write.ErrorID)));
ELSIF _Write.Busy THEN
	PerformAction := OPC_UA_ACTION_EXECUTION_STATE.BUSY;			
END_IF
END_METHOD

METHOD ResetAction
_Write(Execute := FALSE);
END_METHOD

END_FUNCTION_BLOCK

// ---- Communication/OPC_UA/OpcUaHelper.TcPOU
PROGRAM OpcUaHelper
VAR
	ClassName : STRING := __POUNAME();
END_VAR

METHOD GetShortUaIdentifierType : STRING(1)
VAR_INPUT
	identifierType : Tc3_PLCopen_OpcUa.E_UAIdentifierType;
END_VAR
CASE identifierType OF
	Tc3_PLCopen_OpcUa.E_UAIdentifierType.eUAIdentifierType_Numeric:
		GetShortUaIdentifierType := 'i';
		
	Tc3_PLCopen_OpcUa.E_UAIdentifierType.eUAIdentifierType_String:
		GetShortUaIdentifierType := 's';
		
	Tc3_PLCopen_OpcUa.E_UAIdentifierType.eUAIdentifierType_Opaque:
		GetShortUaIdentifierType := 'b';
		
	Tc3_PLCopen_OpcUa.E_UAIdentifierType.eUAIdentifierType_GUID:
		GetShortUaIdentifierType := 'g';
END_CASE
END_METHOD

METHOD ParceStringNodeId : Tc3_PLCopen_OpcUa.ST_UANodeID 
VAR_IN_OUT CONSTANT
	stringNodeId : STRING(1000); // like ns=6;s=Main.WeldConditionController.Configuration
END_VAR
VAR_OUTPUT
	exception : Exception;
END_VAR
VAR
	namespacePart : STRING(10);
	identifierPart : STRING(1000);
	identifierTypePart : STRING(10);
	identifierPathPart : STRING(1000);
END_VAR
IF NOT Tc2_Utilities.FindAndSplitChar(';', ADR(stringNodeId), ADR(namespacePart), SIZEOF(namespacePart), ADR(identifierPart), SIZEOF(identifierPart), FALSE) THEN
	ExceptionHelper.Throw(0, "Symbol ';' is not found in string NodeId representation", __POUNAME(), ClassName, CurrentNamespace.Name, __POSITION());
	RETURN;
END_IF

namespacePart := Tc2_Utilities.F_ToLCase(namespacePart);

IF Tc2_Standard.FIND(namespacePart, 'ns=') <> 1 THEN
	ExceptionHelper.Throw(0, "Sring NodeId should start from 'ns='", __POUNAME(), ClassName, CurrentNamespace.Name, __POSITION());
	RETURN;	
END_IF

namespacePart := Tc2_Standard.DELETE(namespacePart, 3, 1);

ParceStringNodeId.nNamespaceIndex := TO_UINT(namespacePart);

IF NOT Tc2_Utilities.FindAndSplitChar('=', ADR(identifierPart), ADR(identifierTypePart), SIZEOF(identifierTypePart), ADR(identifierPathPart), SIZEOF(identifierPathPart), FALSE) THEN
	ExceptionHelper.Throw(0, "Symbol '=' is not found in string NodeId representation", __POUNAME(), ClassName, CurrentNamespace.Name, __POSITION());
	RETURN;
END_IF

IF identifierPathPart = '' THEN
	ExceptionHelper.Throw(0, "Identifier type is empty", __POUNAME(), ClassName, CurrentNamespace.Name, __POSITION());
	RETURN;	
END_IF

ParceStringNodeId.sIdentifier := identifierPathPart;

IF identifierTypePart = 's' THEN
	ParceStringNodeId.eIdentifierType := Tc3_PLCopen_OpcUa.E_UAIdentifierType.eUAIdentifierType_String;
ELSIF identifierTypePart = 'i' THEN
	ParceStringNodeId.eIdentifierType := Tc3_PLCopen_OpcUa.E_UAIdentifierType.eUAIdentifierType_Numeric;
ELSIF identifierTypePart = 'g' THEN
	ParceStringNodeId.eIdentifierType := Tc3_PLCopen_OpcUa.E_UAIdentifierType.eUAIdentifierType_GUID;
ELSIF identifierTypePart = 'b' THEN
	ParceStringNodeId.eIdentifierType := Tc3_PLCopen_OpcUa.E_UAIdentifierType.eUAIdentifierType_Opaque;
ELSE
	ExceptionHelper.Throw(0, WStringHelper.Concat3("Unknown identifier type '", TO_WSTRING(identifierTypePart), "'"), __POUNAME(), ClassName, CurrentNamespace.Name, __POSITION());
	RETURN;
END_IF
END_METHOD

END_PROGRAM

// ---- Communication/S7/GetStringSizeForS7Comm.TcPOU
FUNCTION GetStringSizeForS7Comm : WORD
VAR_INPUT
	stringVariable : ANY_STRING;
END_VAR

IF stringVariable.diSize < 255 THEN
	GetStringSizeForS7Comm := TO_WORD(stringVariable.diSize);
ELSE
	GetStringSizeForS7Comm := TO_WORD(stringVariable.diSize - 1);
END_IF

END_FUNCTION

// ---- Communication/S7/S7CommunicationSettings.TcPOU
{attribute 'no_explicit_call' := 'do not call this function block directly'} 
FUNCTION_BLOCK S7CommunicationSettings EXTENDS CommunicationSettings
VAR_INPUT
    IpAddrres : STRING(15);
    CpuType : Tc3_S7Comm.E_S7COMM_CPUTYPE;
    Rack : UINT;
    Slot : UINT;
END_VAR
VAR
	_ClassName : STRING := __POUNAME();
END_VAR

PROPERTY CommunicationTypeName : STRING
GET
CommunicationTypeName := 'S7';
END_GET
END_PROPERTY

END_FUNCTION_BLOCK

// ---- Communication/S7/S7Communicator.TcPOU
{attribute 'no_explicit_call' := 'do not call this function block directly'} 
FUNCTION_BLOCK S7Communicator EXTENDS Communicator
VAR
	{attribute 'OPC.UA.DA' := '0'}	
	_ClassName : STRING := __POUNAME();

	{attribute 'OPC.UA.DA' := '0'}	
	_Connection : REFERENCE TO Tc3_S7Comm.FB_S7CommConnection;

	{attribute 'OPC.UA.DA' := '0'}	
	_State : S7_COMMUNICATOR_STATE;
	{attribute 'OPC.UA.DA' := '0'}	
	_DataProcessed : BOOL;
	{attribute 'OPC.UA.DA' := '0'}	
	_Error : BOOL;
	
	{attribute 'OPC.UA.DA' := '0'}	
	_Request : Tc3_S7Comm.FB_S7CommSingleRequest;
	
	{attribute 'OPC.UA.DA' := '0'}	
	_Variables : List(POINTER_TYPE.BYTE_POINTER); // of S7_VARIABLE
	
	{attribute 'OPC.UA.DA' := '0'}	
	_RrequestTimer : Timer;	
END_VAR

METHOD AddRead : BOOL
VAR_INPUT
    targetVariable : ANY;
    byteOffset : WORD;
	bitOffset : BYTE; // ignored for __SYSTEM.__SYSTEM.TYPE_CLASS.TYPE_CLASS.__SYSTEM.TYPE_CLASS.TYPEs other than BOOL
    dataArea : E_S7COMM_DATAAREA;
    dataBlockNumber : WORD;
END_VAR
VAR_OUTPUT
	exception : Exception;
END_VAR
VAR
	result : HRESULT;
END_VAR
CASE targetVariable.TypeClass OF
	__SYSTEM.TYPE_CLASS.TYPE_BOOL:
		result := _Request.AddReadBit(targetVariable.pValue, byteOffset, bitOffset, dataArea, dataBlockNumber);

    __SYSTEM.TYPE_CLASS.TYPE_BIT:
		ExceptionHelper.Throw(0, "BIT data type is not supported. Use BOOL instead", __POUNAME(), ClassName, CurrentNamespace.Name, __POSITION());
		RETURN;
	
    __SYSTEM.TYPE_CLASS.TYPE_BYTE, 
	__SYSTEM.TYPE_CLASS.TYPE_WORD,
    __SYSTEM.TYPE_CLASS.TYPE_DWORD,
    __SYSTEM.TYPE_CLASS.TYPE_LWORD,
    __SYSTEM.TYPE_CLASS.TYPE_SINT,
    __SYSTEM.TYPE_CLASS.TYPE_INT,
    __SYSTEM.TYPE_CLASS.TYPE_DINT,
    __SYSTEM.TYPE_CLASS.TYPE_LINT,
    __SYSTEM.TYPE_CLASS.TYPE_USINT,
    __SYSTEM.TYPE_CLASS.TYPE_UINT,
    __SYSTEM.TYPE_CLASS.TYPE_UDINT,
    __SYSTEM.TYPE_CLASS.TYPE_ULINT,
    __SYSTEM.TYPE_CLASS.TYPE_REAL,
    __SYSTEM.TYPE_CLASS.TYPE_LREAL,
    __SYSTEM.TYPE_CLASS.TYPE_TIME,
    __SYSTEM.TYPE_CLASS.TYPE_DATE,
    __SYSTEM.TYPE_CLASS.TYPE_DATEANDTIME,
    __SYSTEM.TYPE_CLASS.TYPE_TIMEOFDAY,
    __SYSTEM.TYPE_CLASS.TYPE_ENUM,
    __SYSTEM.TYPE_CLASS.TYPE_LTIME:
		result := _Request.AddReadVar(targetVariable.pValue, TO_WORD(targetVariable.diSize), byteOffset, dataArea, dataBlockNumber);

    __SYSTEM.TYPE_CLASS.TYPE_STRING:
		IF targetVariable.diSize < 255 THEN
			result := _Request.AddReadString(targetVariable.pValue, TO_WORD(targetVariable.diSize), byteOffset, dataArea, dataBlockNumber);
		ELSE
			result := _Request.AddReadString(targetVariable.pValue, TO_WORD(targetVariable.diSize - 1), byteOffset, dataArea, dataBlockNumber);
		END_IF
	
    __SYSTEM.TYPE_CLASS.TYPE_WSTRING:
		ExceptionHelper.Throw(0, "WSTRING data type is not supported. Use STRING instead", __POUNAME(), ClassName, CurrentNamespace.Name, __POSITION());
		RETURN;
	
	__SYSTEM.TYPE_CLASS.TYPE_ARRAY:
		result := _Request.AddReadByteArray(targetVariable.pValue, TO_WORD(targetVariable.diSize), byteOffset, dataArea, dataBlockNumber);
	
    ELSE
		ExceptionHelper.Throw(0, WStringHelper.Concat3("Data type ", TO_WSTRING(targetVariable.TypeClass), " is not supported"), __POUNAME(), ClassName, CurrentNamespace.Name, __POSITION());
		RETURN;
END_CASE

CASE result OF
	Tc2_System.E_HRESULTAdsErr.HRESULT_ADS_NOERROR:
		addVariable(targetVariable.pValue, FALSE);
		AddRead := TRUE;
	
	Tc2_System.E_HRESULTAdsErr.NOTINIT:
		ExceptionHelper.Throw(0, "Tc3_S7Comm.FB_S7CommSingleRequest is not initialized correctly", __POUNAME(), ClassName, CurrentNamespace.Name, __POSITION());
	
	Tc2_System.E_HRESULTAdsErr.BUSY:
		ExceptionHelper.Throw(0, "Request is active", __POUNAME(), ClassName, CurrentNamespace.Name, __POSITION());
	
	Tc2_System.E_HRESULTAdsErr.INVALIDDATA:
		ExceptionHelper.Throw(0, "A transfer parameter has been defined incorrectly", __POUNAME(), ClassName, CurrentNamespace.Name, __POSITION());
	
	Tc2_System.E_HRESULTAdsErr.INVALIDSIZE:
		ExceptionHelper.Throw(0, "The frame length is greater than the PDU length", __POUNAME(), ClassName, CurrentNamespace.Name, __POSITION());
		
	ELSE
		ExceptionHelper.Throw(0, WStringHelper.Concat6("Tc3_S7Comm.FB_S7CommSingleRequest method returned HRESULT = ", TO_WSTRING(result), " for byte offset ", TO_WSTRING(byteOffset), " and bit offset ", TO_WSTRING(bitOffset)), __POUNAME(), ClassName, CurrentNamespace.Name, __POSITION());
END_CASE
END_METHOD

METHOD AddReadBit : HRESULT // Try to use AddRead instead
VAR_INPUT
    pVar : PVOID;
    nByteOff : WORD;
    nBitOff : BYTE;
    nArea : E_S7COMM_DATAAREA;
    nDatablock : WORD;
END_VAR
AddReadBit := _Request.AddReadBit(pVar, nByteOff, nBitOff, nArea, nDatablock);

IF AddReadBit = E_HRESULTAdsErr.HRESULT_ADS_NOERROR THEN
	addVariable(pVar, FALSE);
END_IF
END_METHOD

METHOD AddReadByteArray : HRESULT // Try to use AddRead instead
VAR_INPUT
    pVar : PVOID;
    nByteSize : WORD;
    nByteOff : WORD;
    nArea : E_S7COMM_DATAAREA;
    nDatablock : WORD;
END_VAR
AddReadByteArray := _Request.AddReadByteArray(pVar, nByteSize, nByteOff, nArea, nDatablock);

IF AddReadByteArray = E_HRESULTAdsErr.HRESULT_ADS_NOERROR THEN
	addVariable(pVar, FALSE);
END_IF
END_METHOD

METHOD AddReadString : HRESULT // Try to use AddRead instead
VAR_INPUT
    pVar : PVOID;
    nByteSize : WORD;
    nByteOff : WORD;
    nArea : E_S7COMM_DATAAREA;
    nDatablock : WORD;
END_VAR
AddReadString := _Request.AddReadString(pVar, nByteSize, nByteOff, nArea, nDatablock);

IF AddReadString = E_HRESULTAdsErr.HRESULT_ADS_NOERROR THEN
	addVariable(pVar, FALSE);
END_IF
END_METHOD

METHOD AddReadVar : HRESULT // Try to use AddRead instead
VAR_INPUT
    pVar : PVOID;
    nByteSize : WORD;
    nByteOff : WORD;
    nArea : E_S7COMM_DATAAREA;
    nDatablock : WORD;
END_VAR
AddReadVar := _Request.AddReadVar(pVar, nByteSize, nByteOff, nArea, nDatablock);

IF AddReadVar = E_HRESULTAdsErr.HRESULT_ADS_NOERROR THEN
	addVariable(pVar, FALSE);
END_IF
END_METHOD

METHOD PRIVATE addVariable
VAR_INPUT
	address : PVOID;
	write : BOOL;
END_VAR
VAR
	variable : POINTER TO S7_VARIABLE;
END_VAR
variable := __NEW(S7_VARIABLE);

variable^.Address := address;
variable^.Write := write;

_Variables.Append(variable);
END_METHOD

METHOD AddWrite : BOOL
VAR_INPUT
    sourceVariable : ANY;
    byteOffset : WORD;
	bitOffset : BYTE; // ignored for __SYSTEM.__SYSTEM.TYPE_CLASS.TYPE_CLASS.__SYSTEM.TYPE_CLASS.TYPEs other than BOOL
    dataArea : E_S7COMM_DATAAREA;
    dataBlockNumber : WORD;
END_VAR
VAR_OUTPUT
	exception : Exception;
END_VAR
VAR
	result : HRESULT;
END_VAR
CASE sourceVariable.TypeClass OF
	__SYSTEM.TYPE_CLASS.TYPE_BOOL:
		result := _Request.AddWriteBit(sourceVariable.pValue, byteOffset, bitOffset, dataArea, dataBlockNumber);
	
    __SYSTEM.TYPE_CLASS.TYPE_BIT:
		ExceptionHelper.Throw(0, "BIT data type is not supported. Use BOOL instead", __POUNAME(), ClassName, CurrentNamespace.Name, __POSITION());
		RETURN;
	
    __SYSTEM.TYPE_CLASS.TYPE_BYTE, 
	__SYSTEM.TYPE_CLASS.TYPE_WORD,
    __SYSTEM.TYPE_CLASS.TYPE_DWORD,
    __SYSTEM.TYPE_CLASS.TYPE_LWORD,
    __SYSTEM.TYPE_CLASS.TYPE_SINT,
    __SYSTEM.TYPE_CLASS.TYPE_INT,
    __SYSTEM.TYPE_CLASS.TYPE_DINT,
    __SYSTEM.TYPE_CLASS.TYPE_LINT,
    __SYSTEM.TYPE_CLASS.TYPE_USINT,
    __SYSTEM.TYPE_CLASS.TYPE_UINT,
    __SYSTEM.TYPE_CLASS.TYPE_UDINT,
    __SYSTEM.TYPE_CLASS.TYPE_ULINT,
    __SYSTEM.TYPE_CLASS.TYPE_REAL,
    __SYSTEM.TYPE_CLASS.TYPE_LREAL,
    __SYSTEM.TYPE_CLASS.TYPE_TIME,
    __SYSTEM.TYPE_CLASS.TYPE_DATE,
    __SYSTEM.TYPE_CLASS.TYPE_DATEANDTIME,
    __SYSTEM.TYPE_CLASS.TYPE_TIMEOFDAY,
    __SYSTEM.TYPE_CLASS.TYPE_ENUM,
    __SYSTEM.TYPE_CLASS.TYPE_LTIME:
		result := _Request.AddWriteVar(sourceVariable.pValue, TO_WORD(sourceVariable.diSize), byteOffset, dataArea, dataBlockNumber);

    __SYSTEM.TYPE_CLASS.TYPE_STRING:
		IF sourceVariable.diSize < 255 THEN
			result := _Request.AddWriteString(sourceVariable.pValue, TO_WORD(sourceVariable.diSize), byteOffset, dataArea, dataBlockNumber);
		ELSE
			result := _Request.AddWriteString(sourceVariable.pValue, TO_WORD(sourceVariable.diSize - 1), byteOffset, dataArea, dataBlockNumber);
		END_IF
	
    __SYSTEM.TYPE_CLASS.TYPE_WSTRING:
		ExceptionHelper.Throw(0, "WSTRING data type is not supported. Use STRING instead", __POUNAME(), ClassName, CurrentNamespace.Name, __POSITION());
		RETURN;
	
	__SYSTEM.TYPE_CLASS.TYPE_ARRAY:
		result := _Request.AddWriteByteArray(sourceVariable.pValue, TO_WORD(sourceVariable.diSize), byteOffset, dataArea, dataBlockNumber);
	
    ELSE
		ExceptionHelper.Throw(0, WStringHelper.Concat3("Data type ", TO_WSTRING(sourceVariable.TypeClass), " is not supported"), __POUNAME(), ClassName, CurrentNamespace.Name, __POSITION());
		RETURN;
END_CASE

CASE result OF
	Tc2_System.E_HRESULTAdsErr.HRESULT_ADS_NOERROR:
		addVariable(sourceVariable.pValue, TRUE);
		AddWrite := TRUE;
	
	Tc2_System.E_HRESULTAdsErr.NOTINIT:
		ExceptionHelper.Throw(0, "Tc3_S7Comm.FB_S7CommSingleRequest is not initialized correctly", __POUNAME(), ClassName, CurrentNamespace.Name, __POSITION());
	
	Tc2_System.E_HRESULTAdsErr.BUSY:
		ExceptionHelper.Throw(0, "Request is active", __POUNAME(), ClassName, CurrentNamespace.Name, __POSITION());
	
	Tc2_System.E_HRESULTAdsErr.INVALIDDATA:
		ExceptionHelper.Throw(0, "A transfer parameter has been defined incorrectly", __POUNAME(), ClassName, CurrentNamespace.Name, __POSITION());
	
	Tc2_System.E_HRESULTAdsErr.INVALIDSIZE:
		ExceptionHelper.Throw(0, "The frame length is greater than the PDU length", __POUNAME(), ClassName, CurrentNamespace.Name, __POSITION());
		
	ELSE
		ExceptionHelper.Throw(0, WStringHelper.Concat6("Tc3_S7Comm.FB_S7CommSingleRequest method returned HRESULT = ", TO_WSTRING(result), " for byte offset ", TO_WSTRING(byteOffset), " and bit offset ", TO_WSTRING(bitOffset)), __POUNAME(), ClassName, CurrentNamespace.Name, __POSITION());
END_CASE
END_METHOD

METHOD AddWriteBit : HRESULT // try to use AddWrite instead
VAR_INPUT
    pVar : PVOID;
    nByteOff : WORD;
    nBitOff : BYTE;
    nArea : E_S7COMM_DATAAREA;
    nDatablock : WORD;
END_VAR
AddWriteBit := _Request.AddWriteBit(pVar, nByteOff, nBitOff, nArea, nDatablock);

IF AddWriteBit = E_HRESULTAdsErr.HRESULT_ADS_NOERROR THEN
	addVariable(pVar, TRUE);
END_IF
END_METHOD

METHOD AddWriteByteArray : HRESULT
VAR_INPUT
    pVar : PVOID;
    nByteSize : WORD;
    nByteOff : WORD;
    nArea : E_S7COMM_DATAAREA;
    nDatablock : WORD;
END_VAR
AddWriteByteArray := _Request.AddWriteByteArray(pVar, nByteSize, nByteOff, nArea, nDatablock);

IF AddWriteByteArray = E_HRESULTAdsErr.HRESULT_ADS_NOERROR THEN
	addVariable(pVar, TRUE);
END_IF
END_METHOD

METHOD AddWriteString : HRESULT
VAR_INPUT
    pVar : PVOID;
    nByteSize : WORD;
    nByteOff : WORD;
    nArea : E_S7COMM_DATAAREA;
    nDatablock : WORD;
END_VAR
AddWriteString := _Request.AddWriteString(pVar, nByteSize, nByteOff, nArea, nDatablock);

IF AddWriteString = E_HRESULTAdsErr.HRESULT_ADS_NOERROR THEN
	addVariable(pVar, TRUE);
END_IF
END_METHOD

METHOD AddWriteVar : HRESULT
VAR_INPUT
    pVar : PVOID;
    nByteSize : WORD;
    nByteOff : WORD;
    nArea : E_S7COMM_DATAAREA;
    nDatablock : WORD;
END_VAR
AddWriteVar := _Request.AddWriteVar(pVar, nByteSize, nByteOff, nArea, nDatablock);

IF AddWriteVar = E_HRESULTAdsErr.HRESULT_ADS_NOERROR THEN
	addVariable(pVar, TRUE);
END_IF
END_METHOD

{attribute 'monitoring' := 'call'}
{attribute 'OPC.UA.DA' := '1'}
{attribute 'OPC.UA.DA.Property' := '1'}
PROPERTY Busy : BOOL
GET
Busy := _State <> S7_COMMUNICATOR_STATE.IDLE_OR_DONE;
END_GET
END_PROPERTY

{attribute 'monitoring' := 'call'}
PROPERTY ClassName : STRING
GET
ClassName := _ClassName;
END_GET
END_PROPERTY

PROPERTY CommunicationTypeName : STRING
GET
CommunicationTypeName := 'S7';
END_GET
END_PROPERTY

{attribute 'monitoring' := 'call'}
{attribute 'OPC.UA.DA' := '1'}
{attribute 'OPC.UA.DA.Property' := '1'}
PROPERTY DataProcessed : BOOL
GET
DataProcessed := _DataProcessed;
END_GET
END_PROPERTY

{attribute 'monitoring' := 'call'}
{attribute 'OPC.UA.DA' := '1'}
{attribute 'OPC.UA.DA.Property' := '1'}
PROPERTY Error : BOOL
GET
Error := _Error;
END_GET
END_PROPERTY

METHOD Execute
_DataProcessed := FALSE;

_RrequestTimer.Execute();
_Connection();

StateMachine:

CASE _State OF
	S7_COMMUNICATOR_STATE.DATA_PROCESSING:		
		IF _Connection.bIsConnected THEN
			_Request(bExecute := TRUE);
			
			IF _Request.bError THEN
				_State := S7_COMMUNICATOR_STATE.IDLE_OR_DONE;
				_Error := TRUE;
				_LastExceptionHelper.Throw(_Request.nErrorId, TO_WSTRING(_Request.sErrorTxt), __POUNAME(), ClassName, CurrentNamespace.Name, __POSITION());
				
				_Request(bExecute := FALSE);
				_Connection(bExecute := FALSE);
			ELSE
				_DataProcessed := NOT _Request.bBusy;
				_Request(bExecute := FALSE);
				
				IF CyclicMode THEN
					_State := S7_COMMUNICATOR_STATE.WAIT_FOR_NEXT_CYCLE;
					JMP StateMachine;
				ELSE
					_State := S7_COMMUNICATOR_STATE.IDLE_OR_DONE;
				END_IF
			END_IF		
		ELSIF _Connection.bError THEN
			_State := S7_COMMUNICATOR_STATE.IDLE_OR_DONE;
			_Error := TRUE;
			_LastExceptionHelper.Throw(0, TO_WSTRING(_Connection.sErrorTxt), __POUNAME(), ClassName, CurrentNamespace.Name, __POSITION()); 
			
			_Request(bExecute := FALSE);
			_Connection(bExecute := FALSE);
		END_IF	
		
	S7_COMMUNICATOR_STATE.WAIT_FOR_NEXT_CYCLE:
		IF _RrequestTimer.ElapsedTime >= CycleInterval THEN
			_State := S7_COMMUNICATOR_STATE.DATA_PROCESSING;
			JMP StateMachine;			
		END_IF
END_CASE
END_METHOD

METHOD FB_init : BOOL
VAR_INPUT
	bInitRetains : BOOL; // if TRUE, the retain variables are initialized (warm start / cold start)
	bInCopyCode : BOOL;  // if TRUE, the instance afterwards gets moved into the copy code (online change)
	connection : REFERENCE TO Tc3_S7Comm.FB_S7CommConnection;
END_VAR
_Connection REF= connection;
END_METHOD

METHOD PROTECTED InternalClear : BOOL
VAR_OUTPUT
	exception : Exception;
END_VAR
VAR 
	i : DINT;	
	variable : POINTER TO S7_VARIABLE;
END_VAR
FOR i := 0 TO _Variables.Count - 1 DO
	variable := _Variables.Get(i);
	
	IF variable^.Write THEN
		RemoveWrite(variable^.Address);
	ELSE
		RemoveRead(variable^.Address);
	END_IF
END_FOR

_Variables.Clear(TRUE);

_Error := FALSE;

InternalClear := TRUE;
END_METHOD

METHOD PROTECTED InternalConfigure : BOOL
VAR_INPUT
	settings : REFERENCE TO CommunicationSettings;
END_VAR
VAR_OUTPUT
	exception : Exception;
END_VAR
VAR
	s7Settings : POINTER TO S7CommunicationSettings;
END_VAR
IF NOT __ISVALIDREF(_Connection) THEN
	ExceptionHelper.Throw(0, "Connection is null", __POUNAME(), ClassName, CurrentNamespace.Name, __POSITION());
	RETURN;	
END_IF

_RrequestTimer.Interval := T#1H;

//todo: reimplement communication, don't use standard cyclic request
(*IF Configured AND_THEN settings.CyclicMode <> CyclicMode THEN
	ExceptionHelper.Throw(0, "CyclicMode can't be changed fro S7Communicator", "InternalConfigure", ClassName, CurrentNamespace.Name);
	RETURN;		
END_IF*)

s7Settings := ADR(settings);

IF s7Settings^.IpAddrres = '' THEN
	ExceptionHelper.Throw(0, "settings.IpAddrres is empty", __POUNAME(), ClassName, CurrentNamespace.Name, __POSITION());
	RETURN;	
END_IF

_Connection.sIpAddr := s7Settings^.IpAddrres;
_Connection.eCpuType := s7Settings^.CpuType;
_Connection.nRack := s7Settings^.Rack;
_Connection.nSlot := s7Settings^.Slot;

IF NOT Configured THEN
	_Connection.AddRequest(_Request);
END_IF

InternalConfigure := TRUE;
END_METHOD

METHOD PROTECTED InternalStart : BOOL
VAR_OUTPUT
	exception : Exception;
END_VAR
InternalStop();

_Connection(bExecute := TRUE);
_RrequestTimer.Start();

_State := S7_COMMUNICATOR_STATE.DATA_PROCESSING;

InternalStart := TRUE;
END_METHOD

METHOD PROTECTED InternalStop
_Request(bExecute := FALSE);
_Connection(bExecute := FALSE);

_RrequestTimer.Stop();

_State := S7_COMMUNICATOR_STATE.IDLE_OR_DONE;
_Error := FALSE;
END_METHOD

METHOD RemoveRead : HRESULT
VAR_INPUT
    pVar : PVOID;
END_VAR
VAR
	i : DINT;
	variable : POINTER TO S7_VARIABLE;
END_VAR
RemoveRead := _Request.RemoveRead(pVar);

IF RemoveRead = Tc2_System.E_HRESULTAdsErr.HRESULT_ADS_NOERROR THEN
	FOR i := 0 TO _Variables.Count - 1 DO
		variable := _Variables.Get(i);
		
		IF variable^.Address = pVar AND_THEN NOT variable^.Write THEN
			_Variables.Remove(variable, TRUE);		
			RETURN;
		END_IF 
	END_FOR
END_IF
END_METHOD

METHOD RemoveWrite : HRESULT
VAR_INPUT
    pVar : PVOID;
END_VAR
VAR
	i : DINT;
	variable : POINTER TO S7_VARIABLE;
END_VAR
RemoveWrite := _Request.RemoveWrite(pVar);

IF RemoveWrite = Tc2_System.E_HRESULTAdsErr.HRESULT_ADS_NOERROR THEN
	FOR i := 0 TO _Variables.Count - 1 DO
		variable := _Variables.Get(i);
		
		IF variable^.Address = pVar AND_THEN variable^.Write THEN
			_Variables.Remove(variable, TRUE);		
			RETURN;
		END_IF 
	END_FOR
END_IF
END_METHOD

{attribute 'monitoring' := 'call'}
PROPERTY VariablesCount : DINT
GET
VariablesCount := _Variables.Count;
END_GET
END_PROPERTY

END_FUNCTION_BLOCK

// ---- Database/Command/DbCommandExecutor.TcPOU
{attribute 'no_explicit_call' := 'do not call this function block directly'} 
FUNCTION_BLOCK DbCommandExecutor EXTENDS TC.ToolkitObject IMPLEMENTS TC.IAction
VAR	
	_ClassName : STRING := __POUNAME();

	_DbConnection : Tc3_Database.FB_SQLDatabaseEvt(sNetID := '', tTimeout := T#10S);	

	_ExecutionParameters : DB_COMMAND_EXECUTION_PARAMETERS;

	_Command : Tc3_Database.FB_SQLCommandEvt(sNetID:='', tTimeout := T#10S);
	_SQLResult: Tc3_Database.FB_SQLResultEvt(sNetID := '', tTimeout := T#10S);
	
	_Done : BOOL;
	_State : DB_COMMAND_EXECUTION_STATE;
	_GetError : BOOL;
	_Logger : Tc3_EventLogger.I_TcMessage;	
	_Connected : BOOL;
	_DataSetLoaded : BOOL;
	_DisconnectingState : DB_COMMAND_DISCONNECTING_STATE;
	_LastException : Exception;
END_VAR

{attribute 'monitoring' := 'call'}
{attribute 'OPC.UA.DA.Property' := '1'}
{attribute 'OPC.UA.DA.Access' := '1'}
PROPERTY Busy : BOOL
GET
Busy := State <> DB_COMMAND_EXECUTION_STATE.IDLING;
END_GET
END_PROPERTY

{attribute 'monitoring' := 'call'}
PROPERTY ClassName : STRING
GET
ClassName := _ClassName;
END_GET
END_PROPERTY

{attribute 'monitoring' := 'call'}
{attribute 'OPC.UA.DA.Property' := '1'}
{attribute 'OPC.UA.DA.Access' := '1'}
PROPERTY CommandText : REFERENCE TO Tc2_System.T_MaxString
GET
CommandText REF= _ExecutionParameters.CommandText;
END_GET
END_PROPERTY

{attribute 'monitoring' := 'call'}
{attribute 'OPC.UA.DA.Property' := '1'}
{attribute 'OPC.UA.DA.Access' := '1'}
PROPERTY Done : BOOL
GET
Done := _Done;
END_GET
END_PROPERTY

{attribute 'monitoring' := 'call'}
{attribute 'OPC.UA.DA.Property' := '1'}
{attribute 'OPC.UA.DA.Access' := '1'}
PROPERTY Error : BOOL
GET
Error := State = DB_COMMAND_EXECUTION_STATE.IDLING AND_THEN NOT _LastException.Empty;
END_GET
END_PROPERTY

METHOD Execute
VAR
	requestEventTextError : BOOL;	
	requestEventTextErrorCode : HRESULT;
END_VAR
VAR_INST
	errorMessage : STRING(255);	
END_VAR
START:

IF NOT _LastException.Empty THEN
	_GetError := FALSE;
END_IF

IF _GetError THEN
	IF _Logger <> 0 THEN 
		IF _Logger.RequestEventText(1033, errorMessage, SIZEOF(errorMessage), bError => requestEventTextError, hrErrorCode => requestEventTextErrorCode) THEN
			IF requestEventTextError THEN					
				errorMessage := StringHelper.Concat2('_Logger.RequestEventText() call error. Error code is ', TO_STRING(requestEventTextErrorCode));
			END_IF
		ELSE
			RETURN;
		END_IF			
	ELSE
		errorMessage :=  'Logger is not specified';
	END_IF				
	
	_LastExceptionHelper.Throw(0, TO_WSTRING(errorMessage), __POUNAME(), ClassName, CurrentNamespace.Name, __POSITION());
	JMP START;	
END_IF

CASE State OF
	DB_COMMAND_EXECUTION_STATE.STARTING:
		MEMSET(_ExecutionParameters.TargetBuffer, 0, _ExecutionParameters.TargetBufferSize);	
		_State := DB_COMMAND_EXECUTION_STATE.CONNECTING;		
		JMP START;		
	
	DB_COMMAND_EXECUTION_STATE.CONNECTING:
		IF _DbConnection.Connect(hDBID := _ExecutionParameters.DBID) THEN
			IF _DbConnection.bError THEN
				_GetError := TRUE;
				_Logger := _DbConnection.ipTcResult;
				_State := DB_COMMAND_EXECUTION_STATE.DISCONNECTING;				
			ELSE
				_Connected := TRUE;
				_State := DB_COMMAND_EXECUTION_STATE.PREPARING;
			END_IF
			
			JMP START;
		END_IF
	
	DB_COMMAND_EXECUTION_STATE.PREPARING:
		IF _DbConnection.CreateCmd(ADR(_Command)) THEN
			IF _DbConnection.bError THEN
				_GetError := TRUE;
				_Logger := _DbConnection.ipTcResult;
				_State := DB_COMMAND_EXECUTION_STATE.DISCONNECTING;				
			ELSE
				_State := DB_COMMAND_EXECUTION_STATE.EXECUTING;
			END_IF
			
			JMP START;
		END_IF
	
	DB_COMMAND_EXECUTION_STATE.EXECUTING:
		IF _ExecutionParameters.MaxRecordsToReadAtTime = 0 THEN
			IF _Command.Execute(ADR(_ExecutionParameters.CommandText), SIZEOF(_ExecutionParameters.CommandText)) THEN
				IF _Command.bError THEN
					_GetError := TRUE;
					_Logger := _Command.ipTcResult;
				END_IF
				
				_State := DB_COMMAND_EXECUTION_STATE.DISCONNECTING;
				
